(* CoDeSys 2.3.9.41 project: GermesLib_1_51.pro *)
(* Libraries: PID_Regulators.lib 6.11.19 15:29:27, Util.lib 18.5.10 15:14:28, STANDARD.LIB 4.10.05 11:14:46, IECSFC.LIB 13.4.06 15:51:28, ANALYZATION.LIB 5.10.99 09:05:06 *)

(* PLC configuration (modules and I/O channels)
Fast discrete inputs [I_SIMPLE_INPUT] node 0, in %IB0 out %QB0 {Filtrationtime = 10}
  DD1_DI0 AT %IX0.0 [BitInput] резерв
  DD1_DI1 AT %IX0.1 [BitInput] резерв
  DD1_DI2 AT %IX0.2 [BitInput] резерв
  DD1_DI3 AT %IX0.3 [BitInput] резерв
Discrete inputs [ID130] node 1, in %IB1 out %QB1 {Filtrationtime_GeneralINP = 10; Visibility = No; PinCount = 12}
  AT %IB1.0 [ByteInput] 8 discrete inputs
  AT %IB1.1 [ByteInput] 4 discrete inputs
Discrete outputs [ID131] node 2, in %IB2 out %QB2 {SafeValueByte = 0; SafeValueByteM = 0; Visibility = No; PinCount = 12}
  AT %QB2.0 [ByteOutput] 8 discrete outputs
  AT %QB2.1 [ByteOutput] 4 discrete outputs
Fast analog inputs [ID125] node 3, in %IB3 out %QB3 {Flt_Comm = 50Hz 2Por}
  DD1_AI0 AT %IR3.0 [FloatInputP] AI #1 - датчик температуры в помещении (метран) {AIN_TYPE = 4-20 mA; Peak_Filtr = 200; Flt_Ch = Off; TauRC = 10; MinFV = 0; MaxFV = 100}
  DD1_AI1 AT %IR3.1 [FloatInputP] AI #2 - расходомер FT01.01 (на входе, до отстойника) {AIN_TYPE = 4-20 mA; Peak_Filtr = 200; Flt_Ch = Off; TauRC = 10; MinFV = 0; MaxFV = 600}
  DD1_AI2 AT %IR3.2 [FloatInputP] AI #3 - расходомер FT01.02 (на выходе, после отстойника) {AIN_TYPE = 4-20 mA; Peak_Filtr = 200; Flt_Ch = Off; TauRC = 10; MinFV = 0; MaxFV = 600}
  DD1_AI3 AT %IR3.3 [FloatInputP] AI #4 - рН-метр QE01.01 (на входе, до отстойника) {AIN_TYPE = 4-20 mA; Peak_Filtr = 200; Flt_Ch = Off; TauRC = 10; MinFV = 0; MaxFV = 14}
  DD1_AI4 AT %IR3.4 [FloatInputP] AI #5 - рН-метр QE01.02 (на выходе, после отстойника) {AIN_TYPE = 4-20 mA; Peak_Filtr = 200; Flt_Ch = Off; TauRC = 10; MinFV = 0; MaxFV = 14}
  DD1_AI5 AT %IR3.5 [FloatInputP] AI #6 - сигнал от ФПК, давление на входе {AIN_TYPE = 4-20 mA; Peak_Filtr = 200; Flt_Ch = Off; TauRC = 10; MinFV = 0; MaxFV = 16}
  DD1_AI6 AT %IR3.6 [FloatInputP] AI #7 - резерв {AIN_TYPE = 4-20 mA; Peak_Filtr = 200; Flt_Ch = Off; TauRC = 10; MinFV = 0; MaxFV = 20000.0}
  DD1_AI7 AT %IR3.7 [FloatInputP] AI#8 - резерв {AIN_TYPE = 4-20 mA; Peak_Filtr = 200; Flt_Ch = Off; TauRC = 10; MinFV = 0; MaxFV = 20000.0}
  AT %IW3.8 [WordInput] AI read time (10ms)
Analog outputs [ID126] node 4, in %IB4 out %QB4
  DD1_AO0 AT %QR4.0 [FloatOutputP] AO #1 - управление ЧРП Н01.05 (поддержание расхода по расходомеру FT01.02) {AOUT_TYPE = 4-20 mA; SafeValueREAL = 0.0}
  DD1_AO1 AT %QR4.1 [FloatOutputP] AO #2 - управление ЧРП НД08.03/01 (подача флокулянта на входе, до отстойника, по FT01.01) {AOUT_TYPE = 4-20 mA; SafeValueREAL = 0.0}
  DD1_AO2 AT %QR4.2 [FloatOutputP] AO #3 - управление ЧРП НД08.03/02 (подача флокулянта на входе, до отстойника, по FT01.01) {AOUT_TYPE = 4-20 mA; SafeValueREAL = 0.0}
  DD1_AO3 AT %QR4.3 [FloatOutputP] AO #4 - управление НД05.02/01 (подача 10%NaCl из УПГ на входе, до отстойника, по FT01.01) {AOUT_TYPE = 4-20 mA; SafeValueREAL = 0.0}
Special input [ID103] node 5, in %IB5 out %QB5 {Filtrationtime = 1000; PinCount = 1; WatchDogPeriod = 400; PollPeriod = 3000; Visibility = No}
  AT %IX5.0 [BitInput] Special input
Special output [ID104] node 6, in %IB6 out %QB6 {Visibility = No; PinCount = 1}
  AT %QX6.0 [BitOutput] Special output
lastAddress AT %QD7.0 [DWordOutput] Last address
lastError AT %QW7.1 [WordOutput] Last error
RS-485-1 [COM1_USART] node 0, in %IB7.0 out %QB7.0 {CommunicationSpeed = 9600; Parity = EVEN; BitLength = 8 bits; StopLength = One stop bit; InterfaceType = RS485; FrameOriented = RTU; Timeout = 0; Visibility = No}
Universal Modbus device [ID2000] node 1, in %IB7.1 out %QB7.1 {ModuleIP = 10:0:0:102; ServiceTimeout = 20; TCPport = 502; NetMode = Serial; ModuleSlaveAddress = 2; RequestType = Both; PeriodOfService = 100; Visibility = No; RepeatCounter = 0; ByteSequence = Trace_mode}
  AT %QB7.1.0 [ComChannel] Command (0xff - Start)
DD2_DO AT %QD7.1.0.0 [DWordOutput] регистр 0, команда 0х0f
Universal Modbus device [ID2000] node 2, in %IB7.2 out %QB7.2 {ModuleIP = 10:0:0:103; ServiceTimeout = 20; TCPport = 502; NetMode = Serial; ModuleSlaveAddress = 3; RequestType = Both; PeriodOfService = 100; Visibility = No; RepeatCounter = 0; ByteSequence = Trace_mode}
  AT %QB7.2.0 [ComChannel] Command (0xff - Start)
DD3_DO AT %QD7.2.0.0 [DWordOutput]
Universal Modbus device [ID2000] node 3, in %IB7.3 out %QB7.3 {ModuleIP = 10:0:0:104; ServiceTimeout = 20; TCPport = 502; NetMode = Serial; ModuleSlaveAddress = 4; RequestType = Both; PeriodOfService = 100; Visibility = No; RepeatCounter = 0; ByteSequence = Trace_mode}
  AT %QB7.3.0 [ComChannel] Command (0xff - Start)
  32bit output module [ID2006] node 0, in %IB7.3.0 out %QB7.3.0 {ModbusAddress = 0; Command_write_regs = Force multiple coils (0x0f); Visibility = No}
    DD4_DO AT %QD7.3.0.0 [DWordOutput]
Universal Modbus device [ID2000] node 4, in %IB7.4 out %QB7.4 {ModuleIP = 10:0:0:105; ServiceTimeout = 20; TCPport = 502; NetMode = Serial; ModuleSlaveAddress = 5; RequestType = Both; PeriodOfService = 100; Visibility = No; RepeatCounter = 0; ByteSequence = Trace_mode}
  AT %QB7.4.0 [ComChannel] Command (0xff - Start)
DD5_DI AT %ID7.4.0.0 [DWordInput]
Universal Modbus device [ID2000] node 5, in %IB7.5 out %QB7.5 {ModuleIP = 10:0:0:106; ServiceTimeout = 20; TCPport = 502; NetMode = Serial; ModuleSlaveAddress = 6; RequestType = Both; PeriodOfService = 100; Visibility = No; RepeatCounter = 0; ByteSequence = Trace_mode}
  AT %QB7.5.0 [ComChannel] Command (0xff - Start)
DD6_DI AT %ID7.5.0.0 [DWordInput]
Universal Modbus device [ID2000] node 6, in %IB7.6 out %QB7.6 {ModuleIP = 10:0:0:107; ServiceTimeout = 20; TCPport = 502; NetMode = Serial; ModuleSlaveAddress = 7; RequestType = Both; PeriodOfService = 100; Visibility = No; RepeatCounter = 0; ByteSequence = Trace_mode}
  AT %QB7.6.0 [ComChannel] Command (0xff - Start)
DD7_DI AT %ID7.6.0.0 [DWordInput]
Universal Modbus device [ID2000] node 7, in %IB7.7 out %QB7.7 {ModuleIP = 10:0:0:108; ServiceTimeout = 20; TCPport = 502; NetMode = Serial; ModuleSlaveAddress = 8; RequestType = Both; PeriodOfService = 100; Visibility = No; RepeatCounter = 0; ByteSequence = Trace_mode}
  AT %QB7.7.0 [ComChannel] Command (0xff - Start)
DD8_DI AT %ID7.7.0.0 [DWordInput]
Universal Modbus device [ID2000] node 8, in %IB7.8 out %QB7.8 {ModuleIP = 10:0:0:109; ServiceTimeout = 20; TCPport = 502; NetMode = Serial; ModuleSlaveAddress = 9; RequestType = Both; PeriodOfService = 100; Visibility = No; RepeatCounter = 0; ByteSequence = Trace_mode}
  AT %QB7.8.0 [ComChannel] Command (0xff - Start)
DD9_DI AT %ID7.8.0.0 [DWordInput]
Universal Modbus device [ID2000] node 9, in %IB7.9 out %QB7.9 {ModuleIP = 10:0:0:110; ServiceTimeout = 20; TCPport = 502; NetMode = Serial; ModuleSlaveAddress = 10; RequestType = Both; PeriodOfService = 100; Visibility = No; RepeatCounter = 0; ByteSequence = Trace_mode}
  AT %QB7.9.0 [ComChannel] Command (0xff - Start)
DD10_AO0 AT %QW7.9.0.0 [WordOutput] управление 4...20мА НД05.02/02
DD10_AO1 AT %QW7.9.1.0 [WordOutput] управление 4...20мА НД06.02/01
DD10_AO2 AT %QW7.9.2.0 [WordOutput] управление 4...20мА НД06.02/02
DD10_AO3 AT %QW7.9.3.0 [WordOutput] управление 4...20мА НД06.03/01
DD10_AO4 AT %QW7.9.4.0 [WordOutput] управление 4...20мА НД06.03/02
DD10_AO5 AT %QW7.9.5.0 [WordOutput] управление 4...20мА НД07.03/01
DD10_AO6 AT %QW7.9.6.0 [WordOutput] управление 4...20мА НД07.03/02
DD10_AO7 AT %QW7.9.7.0 [WordOutput] управление 4...20мА НД08.04
Universal Modbus device [ID2000] node 10, in %IB7.10 out %QB7.10 {ModuleIP = 10:0:0:223; ServiceTimeout = 20; TCPport = 502; NetMode = Serial; ModuleSlaveAddress = 11; RequestType = By value change; PeriodOfService = 100; Visibility = No; RepeatCounter = 0; ByteSequence = Trace_mode}
  AT %QB7.10.0 [ComChannel] Command (0xff - Start)
AT %QB7.10.0.0 [ByteOutput]
Universal Modbus device [ID2000] node 11, in %IB7.11 out %QB7.11 {ModuleIP = 10:0:0:223; ServiceTimeout = 20; TCPport = 502; NetMode = Serial; ModuleSlaveAddress = 11; RequestType = By poll time; PeriodOfService = 100; Visibility = No; RepeatCounter = 0; ByteSequence = Trace_mode}
  AT %QB7.11.0 [ComChannel] Command (0xff - Start)
AT %IB7.11.0.0 [ByteInput]
Universal Modbus device [ID2000] node 12, in %IB7.12 out %QB7.12 {ModuleIP = 10:0:0:223; ServiceTimeout = 20; TCPport = 502; NetMode = Serial; ModuleSlaveAddress = 12; RequestType = By value change; PeriodOfService = 100; Visibility = No; RepeatCounter = 0; ByteSequence = Trace_mode}
  AT %QB7.12.0 [ComChannel] Command (0xff - Start)
AT %QB7.12.0.0 [ByteOutput]
Universal Modbus device [ID2000] node 13, in %IB7.13 out %QB7.13 {ModuleIP = 10:0:0:223; ServiceTimeout = 20; TCPport = 502; NetMode = Serial; ModuleSlaveAddress = 12; RequestType = By poll time; PeriodOfService = 100; Visibility = No; RepeatCounter = 0; ByteSequence = Trace_mode}
  AT %QB7.13.0 [ComChannel] Command (0xff - Start)
AT %IB7.13.0.0 [ByteInput]
AT %QD8.0 [DWordOutput] Last address
AT %QW8.1 [WordOutput] Last error
RS-232 [COM2_USART] node 0, in %IB8.0 out %QB8.0 {CommunicationSpeed = 57600; Parity = NO PARITY CHECK; BitLength = 8 bits; StopLength = One stop bit; InterfaceType = RS232; FrameOriented = RTU; Timeout = 0; Visibility = No}
AT %QB8.1.0 [ComChannel] Command (0xff - Start)
Real output module [ID2008] node 0, in %IB8.1.0 out %QB8.1.0 {ModbusAddress = 256; Command_write_regs = Preset multiple Registers (0x10); Visibility = No}
  panFT0101value AT %QD8.1.0.0 [FloatOutput]
Real output module [ID2008] node 1, in %IB8.1.1 out %QB8.1.1 {ModbusAddress = 258; Command_write_regs = Preset multiple Registers (0x10); Visibility = No}
  panQE0101value AT %QD8.1.1.0 [FloatOutput]
Real output module [ID2008] node 2, in %IB8.1.2 out %QB8.1.2 {ModbusAddress = 260; Command_write_regs = Preset multiple Registers (0x10); Visibility = No}
  panFT0102value AT %QD8.1.2.0 [FloatOutput]
Real output module [ID2008] node 3, in %IB8.1.3 out %QB8.1.3 {ModbusAddress = 262; Command_write_regs = Preset multiple Registers (0x10); Visibility = No}
  panQE0102value AT %QD8.1.3.0 [FloatOutput]
Real output module [ID2008] node 4, in %IB8.1.4 out %QB8.1.4 {ModbusAddress = 264; Command_write_regs = Preset multiple Registers (0x10); Visibility = No}
  panFPKpressureValue AT %QD8.1.4.0 [FloatOutput]
Real output module [ID2008] node 5, in %IB8.1.5 out %QB8.1.5 {ModbusAddress = 266; Command_write_regs = Preset multiple Registers (0x10); Visibility = No}
  panFQS0301total AT %QD8.1.5.0 [FloatOutput]
Real output module [ID2008] node 6, in %IB8.1.6 out %QB8.1.6 {ModbusAddress = 268; Command_write_regs = Preset multiple Registers (0x10); Visibility = No}
  panTemperature AT %QD8.1.6.0 [FloatOutput]
Register output module [ID2004] node 7, in %IB8.1.7 out %QB8.1.7 {ModbusAddress = 270; Command_write_one_reg = Write multiple registers(0x10); Visibility = No}
  panND050201workDays AT %QW8.1.7.0 [WordOutput]
Register output module [ID2004] node 8, in %IB8.1.8 out %QB8.1.8 {ModbusAddress = 271; Command_write_one_reg = Write multiple registers(0x10); Visibility = No}
  panND050201workHours AT %QW8.1.8.0 [WordOutput]
Register output module [ID2004] node 9, in %IB8.1.9 out %QB8.1.9 {ModbusAddress = 272; Command_write_one_reg = Write multiple registers(0x10); Visibility = No}
  panND050201workMinutes AT %QW8.1.9.0 [WordOutput]
Register output module [ID2004] node 10, in %IB8.1.10 out %QB8.1.10 {ModbusAddress = 273; Command_write_one_reg = Write multiple registers(0x10); Visibility = No}
  panND050201workSeconds AT %QW8.1.10.0 [WordOutput]
Register output module [ID2004] node 11, in %IB8.1.11 out %QB8.1.11 {ModbusAddress = 274; Command_write_one_reg = Write multiple registers(0x10); Visibility = No}
  panND050202workDays AT %QW8.1.11.0 [WordOutput]
Register output module [ID2004] node 12, in %IB8.1.12 out %QB8.1.12 {ModbusAddress = 275; Command_write_one_reg = Write multiple registers(0x10); Visibility = No}
  panND050202workHours AT %QW8.1.12.0 [WordOutput]
Register output module [ID2004] node 13, in %IB8.1.13 out %QB8.1.13 {ModbusAddress = 276; Command_write_one_reg = Write multiple registers(0x10); Visibility = No}
  panND050202workMinutes AT %QW8.1.13.0 [WordOutput]
Register output module [ID2004] node 14, in %IB8.1.14 out %QB8.1.14 {ModbusAddress = 277; Command_write_one_reg = Write multiple registers(0x10); Visibility = No}
  panND050202workSeconds AT %QW8.1.14.0 [WordOutput]
Register output module [ID2004] node 15, in %IB8.1.15 out %QB8.1.15 {ModbusAddress = 278; Command_write_one_reg = Write multiple registers(0x10); Visibility = No}
  panND0502counterP1 AT %QW8.1.15.0 [WordOutput]
Register output module [ID2004] node 16, in %IB8.1.16 out %QB8.1.16 {ModbusAddress = 279; Command_write_one_reg = Write multiple registers(0x10); Visibility = No}
  panND0502counterP2 AT %QW8.1.16.0 [WordOutput]
Register output module [ID2004] node 17, in %IB8.1.17 out %QB8.1.17 {ModbusAddress = 280; Command_write_one_reg = Write multiple registers(0x10); Visibility = No}
  panND060201workDays AT %QW8.1.17.0 [WordOutput]
Register output module [ID2004] node 18, in %IB8.1.18 out %QB8.1.18 {ModbusAddress = 281; Command_write_one_reg = Write multiple registers(0x10); Visibility = No}
  panND060201workHours AT %QW8.1.18.0 [WordOutput]
Register output module [ID2004] node 19, in %IB8.1.19 out %QB8.1.19 {ModbusAddress = 282; Command_write_one_reg = Write multiple registers(0x10); Visibility = No}
  panND060201workMinutes AT %QW8.1.19.0 [WordOutput]
Register output module [ID2004] node 20, in %IB8.1.20 out %QB8.1.20 {ModbusAddress = 283; Command_write_one_reg = Write multiple registers(0x10); Visibility = No}
  panND060201workSeconds AT %QW8.1.20.0 [WordOutput]
Register output module [ID2004] node 21, in %IB8.1.21 out %QB8.1.21 {ModbusAddress = 284; Command_write_one_reg = Write multiple registers(0x10); Visibility = No}
  panND060202workDays AT %QW8.1.21.0 [WordOutput]
Register output module [ID2004] node 22, in %IB8.1.22 out %QB8.1.22 {ModbusAddress = 285; Command_write_one_reg = Write multiple registers(0x10); Visibility = No}
  panND060202workHours AT %QW8.1.22.0 [WordOutput]
Register output module [ID2004] node 23, in %IB8.1.23 out %QB8.1.23 {ModbusAddress = 286; Command_write_one_reg = Write multiple registers(0x10); Visibility = No}
  panND060202workMinutes AT %QW8.1.23.0 [WordOutput]
Register output module [ID2004] node 24, in %IB8.1.24 out %QB8.1.24 {ModbusAddress = 287; Command_write_one_reg = Write multiple registers(0x10); Visibility = No}
  panND060202workSeconds AT %QW8.1.24.0 [WordOutput]
Register output module [ID2004] node 25, in %IB8.1.25 out %QB8.1.25 {ModbusAddress = 288; Command_write_one_reg = Write multiple registers(0x10); Visibility = No}
  panND0602counterP1 AT %QW8.1.25.0 [WordOutput]
Register output module [ID2004] node 26, in %IB8.1.26 out %QB8.1.26 {ModbusAddress = 289; Command_write_one_reg = Write multiple registers(0x10); Visibility = No}
  panND0602counterP2 AT %QW8.1.26.0 [WordOutput]
Register output module [ID2004] node 27, in %IB8.1.27 out %QB8.1.27 {ModbusAddress = 290; Command_write_one_reg = Write multiple registers(0x10); Visibility = No}
  panND060301workDays AT %QW8.1.27.0 [WordOutput]
Register output module [ID2004] node 28, in %IB8.1.28 out %QB8.1.28 {ModbusAddress = 291; Command_write_one_reg = Write multiple registers(0x10); Visibility = No}
  panND060301workHours AT %QW8.1.28.0 [WordOutput]
Register output module [ID2004] node 29, in %IB8.1.29 out %QB8.1.29 {ModbusAddress = 292; Command_write_one_reg = Write multiple registers(0x10); Visibility = No}
  panND060301workMinutes AT %QW8.1.29.0 [WordOutput]
Register output module [ID2004] node 30, in %IB8.1.30 out %QB8.1.30 {ModbusAddress = 293; Command_write_one_reg = Write multiple registers(0x10); Visibility = No}
  panND060301workSeconds AT %QW8.1.30.0 [WordOutput]
Register output module [ID2004] node 31, in %IB8.1.31 out %QB8.1.31 {ModbusAddress = 294; Command_write_one_reg = Write multiple registers(0x10); Visibility = No}
  panND060302workDays AT %QW8.1.31.0 [WordOutput]
Register output module [ID2004] node 32, in %IB8.1.32 out %QB8.1.32 {ModbusAddress = 295; Command_write_one_reg = Write multiple registers(0x10); Visibility = No}
  panND060302workHours AT %QW8.1.32.0 [WordOutput]
Register output module [ID2004] node 33, in %IB8.1.33 out %QB8.1.33 {ModbusAddress = 296; Command_write_one_reg = Write multiple registers(0x10); Visibility = No}
  panND060302workMinutes AT %QW8.1.33.0 [WordOutput]
Register output module [ID2004] node 34, in %IB8.1.34 out %QB8.1.34 {ModbusAddress = 297; Command_write_one_reg = Write multiple registers(0x10); Visibility = No}
  panND060302workSeconds AT %QW8.1.34.0 [WordOutput]
Register output module [ID2004] node 35, in %IB8.1.35 out %QB8.1.35 {ModbusAddress = 298; Command_write_one_reg = Write multiple registers(0x10); Visibility = No}
  panND0603counterP1 AT %QW8.1.35.0 [WordOutput]
Register output module [ID2004] node 36, in %IB8.1.36 out %QB8.1.36 {ModbusAddress = 299; Command_write_one_reg = Write multiple registers(0x10); Visibility = No}
  panND0603counterP2 AT %QW8.1.36.0 [WordOutput]
Register output module [ID2004] node 37, in %IB8.1.37 out %QB8.1.37 {ModbusAddress = 300; Command_write_one_reg = Write multiple registers(0x10); Visibility = No}
  panND070301workDays AT %QW8.1.37.0 [WordOutput]
Register output module [ID2004] node 38, in %IB8.1.38 out %QB8.1.38 {ModbusAddress = 301; Command_write_one_reg = Write multiple registers(0x10); Visibility = No}
  panND070301workHours AT %QW8.1.38.0 [WordOutput]
Register output module [ID2004] node 39, in %IB8.1.39 out %QB8.1.39 {ModbusAddress = 302; Command_write_one_reg = Write multiple registers(0x10); Visibility = No}
  panND070301workMinutes AT %QW8.1.39.0 [WordOutput]
Register output module [ID2004] node 40, in %IB8.1.40 out %QB8.1.40 {ModbusAddress = 303; Command_write_one_reg = Write multiple registers(0x10); Visibility = No}
  panND070301workSeconds AT %QW8.1.40.0 [WordOutput]
Register output module [ID2004] node 41, in %IB8.1.41 out %QB8.1.41 {ModbusAddress = 304; Command_write_one_reg = Write multiple registers(0x10); Visibility = No}
  panND070302workDays AT %QW8.1.41.0 [WordOutput]
Register output module [ID2004] node 42, in %IB8.1.42 out %QB8.1.42 {ModbusAddress = 305; Command_write_one_reg = Write multiple registers(0x10); Visibility = No}
  panND070302workHours AT %QW8.1.42.0 [WordOutput]
Register output module [ID2004] node 43, in %IB8.1.43 out %QB8.1.43 {ModbusAddress = 306; Command_write_one_reg = Write multiple registers(0x10); Visibility = No}
  panND070302workMinutes AT %QW8.1.43.0 [WordOutput]
Register output module [ID2004] node 44, in %IB8.1.44 out %QB8.1.44 {ModbusAddress = 307; Command_write_one_reg = Write multiple registers(0x10); Visibility = No}
  panND070302workSeconds AT %QW8.1.44.0 [WordOutput]
Register output module [ID2004] node 45, in %IB8.1.45 out %QB8.1.45 {ModbusAddress = 308; Command_write_one_reg = Write multiple registers(0x10); Visibility = No}
  panND0703counterP1 AT %QW8.1.45.0 [WordOutput]
Register output module [ID2004] node 46, in %IB8.1.46 out %QB8.1.46 {ModbusAddress = 309; Command_write_one_reg = Write multiple registers(0x10); Visibility = No}
  panND0703counterP2 AT %QW8.1.46.0 [WordOutput]
Register output module [ID2004] node 47, in %IB8.1.47 out %QB8.1.47 {ModbusAddress = 310; Command_write_one_reg = Write multiple registers(0x10); Visibility = No}
  panND080301workDays AT %QW8.1.47.0 [WordOutput]
Register output module [ID2004] node 48, in %IB8.1.48 out %QB8.1.48 {ModbusAddress = 311; Command_write_one_reg = Write multiple registers(0x10); Visibility = No}
  panND080301workHours AT %QW8.1.48.0 [WordOutput]
Register output module [ID2004] node 49, in %IB8.1.49 out %QB8.1.49 {ModbusAddress = 312; Command_write_one_reg = Write multiple registers(0x10); Visibility = No}
  panND080301workMinutes AT %QW8.1.49.0 [WordOutput]
Register output module [ID2004] node 50, in %IB8.1.50 out %QB8.1.50 {ModbusAddress = 313; Command_write_one_reg = Write multiple registers(0x10); Visibility = No}
  panND080301workSeconds AT %QW8.1.50.0 [WordOutput]
Register output module [ID2004] node 51, in %IB8.1.51 out %QB8.1.51 {ModbusAddress = 314; Command_write_one_reg = Write multiple registers(0x10); Visibility = No}
  panND080302workDays AT %QW8.1.51.0 [WordOutput]
Register output module [ID2004] node 52, in %IB8.1.52 out %QB8.1.52 {ModbusAddress = 315; Command_write_one_reg = Write multiple registers(0x10); Visibility = No}
  panND080302workHours AT %QW8.1.52.0 [WordOutput]
Register output module [ID2004] node 53, in %IB8.1.53 out %QB8.1.53 {ModbusAddress = 316; Command_write_one_reg = Write multiple registers(0x10); Visibility = No}
  panND080302workMinutes AT %QW8.1.53.0 [WordOutput]
Register output module [ID2004] node 54, in %IB8.1.54 out %QB8.1.54 {ModbusAddress = 317; Command_write_one_reg = Write multiple registers(0x10); Visibility = No}
  panND080302workSeconds AT %QW8.1.54.0 [WordOutput]
Register output module [ID2004] node 55, in %IB8.1.55 out %QB8.1.55 {ModbusAddress = 318; Command_write_one_reg = Write multiple registers(0x10); Visibility = No}
  panND0803counterP1 AT %QW8.1.55.0 [WordOutput]
Register output module [ID2004] node 56, in %IB8.1.56 out %QB8.1.56 {ModbusAddress = 319; Command_write_one_reg = Write multiple registers(0x10); Visibility = No}
  panND0803counterP2 AT %QW8.1.56.0 [WordOutput]
Register output module [ID2004] node 57, in %IB8.1.57 out %QB8.1.57 {ModbusAddress = 320; Command_write_one_reg = Write multiple registers(0x10); Visibility = No}
  panN010501workDays AT %QW8.1.57.0 [WordOutput]
Register output module [ID2004] node 58, in %IB8.1.58 out %QB8.1.58 {ModbusAddress = 321; Command_write_one_reg = Write multiple registers(0x10); Visibility = No}
  panN010501workHours AT %QW8.1.58.0 [WordOutput]
Register output module [ID2004] node 59, in %IB8.1.59 out %QB8.1.59 {ModbusAddress = 322; Command_write_one_reg = Write multiple registers(0x10); Visibility = No}
  panN010501workMinutes AT %QW8.1.59.0 [WordOutput]
Register output module [ID2004] node 60, in %IB8.1.60 out %QB8.1.60 {ModbusAddress = 323; Command_write_one_reg = Write multiple registers(0x10); Visibility = No}
  panN010501workSeconds AT %QW8.1.60.0 [WordOutput]
Register output module [ID2004] node 61, in %IB8.1.61 out %QB8.1.61 {ModbusAddress = 324; Command_write_one_reg = Write multiple registers(0x10); Visibility = No}
  panN010502workDays AT %QW8.1.61.0 [WordOutput]
Register output module [ID2004] node 62, in %IB8.1.62 out %QB8.1.62 {ModbusAddress = 325; Command_write_one_reg = Write multiple registers(0x10); Visibility = No}
  panN010502workHours AT %QW8.1.62.0 [WordOutput]
Register output module [ID2004] node 63, in %IB8.1.63 out %QB8.1.63 {ModbusAddress = 326; Command_write_one_reg = Write multiple registers(0x10); Visibility = No}
  panN010502workMinutes AT %QW8.1.63.0 [WordOutput]
Register output module [ID2004] node 64, in %IB8.1.64 out %QB8.1.64 {ModbusAddress = 327; Command_write_one_reg = Write multiple registers(0x10); Visibility = No}
  panN010502workSeconds AT %QW8.1.64.0 [WordOutput]
Register output module [ID2004] node 65, in %IB8.1.65 out %QB8.1.65 {ModbusAddress = 328; Command_write_one_reg = Write multiple registers(0x10); Visibility = No}
  panN0105counterP1 AT %QW8.1.65.0 [WordOutput]
Register output module [ID2004] node 66, in %IB8.1.66 out %QB8.1.66 {ModbusAddress = 329; Command_write_one_reg = Write multiple registers(0x10); Visibility = No}
  panN0105counterP2 AT %QW8.1.66.0 [WordOutput]
Register output module [ID2004] node 67, in %IB8.1.67 out %QB8.1.67 {ModbusAddress = 330; Command_write_one_reg = Write multiple registers(0x10); Visibility = No}
  panN020401workDays AT %QW8.1.67.0 [WordOutput]
Register output module [ID2004] node 68, in %IB8.1.68 out %QB8.1.68 {ModbusAddress = 331; Command_write_one_reg = Write multiple registers(0x10); Visibility = No}
  panN020401workHours AT %QW8.1.68.0 [WordOutput]
Register output module [ID2004] node 69, in %IB8.1.69 out %QB8.1.69 {ModbusAddress = 332; Command_write_one_reg = Write multiple registers(0x10); Visibility = No}
  panN020401workMinutes AT %QW8.1.69.0 [WordOutput]
Register output module [ID2004] node 70, in %IB8.1.70 out %QB8.1.70 {ModbusAddress = 333; Command_write_one_reg = Write multiple registers(0x10); Visibility = No}
  panN020401workSeconds AT %QW8.1.70.0 [WordOutput]
Register output module [ID2004] node 71, in %IB8.1.71 out %QB8.1.71 {ModbusAddress = 334; Command_write_one_reg = Write multiple registers(0x10); Visibility = No}
  panN020402workDays AT %QW8.1.71.0 [WordOutput]
Register output module [ID2004] node 72, in %IB8.1.72 out %QB8.1.72 {ModbusAddress = 335; Command_write_one_reg = Write multiple registers(0x10); Visibility = No}
  panN020402workHours AT %QW8.1.72.0 [WordOutput]
Register output module [ID2004] node 73, in %IB8.1.73 out %QB8.1.73 {ModbusAddress = 336; Command_write_one_reg = Write multiple registers(0x10); Visibility = No}
  panN020402workMinutes AT %QW8.1.73.0 [WordOutput]
Register output module [ID2004] node 74, in %IB8.1.74 out %QB8.1.74 {ModbusAddress = 337; Command_write_one_reg = Write multiple registers(0x10); Visibility = No}
  panN020402workSeconds AT %QW8.1.74.0 [WordOutput]
Register output module [ID2004] node 75, in %IB8.1.75 out %QB8.1.75 {ModbusAddress = 338; Command_write_one_reg = Write multiple registers(0x10); Visibility = No}
  panN0204counterP1 AT %QW8.1.75.0 [WordOutput]
Register output module [ID2004] node 76, in %IB8.1.76 out %QB8.1.76 {ModbusAddress = 339; Command_write_one_reg = Write multiple registers(0x10); Visibility = No}
  panN0204counterP2 AT %QW8.1.76.0 [WordOutput]
Register output module [ID2004] node 77, in %IB8.1.77 out %QB8.1.77 {ModbusAddress = 340; Command_write_one_reg = Write multiple registers(0x10); Visibility = No}
  panN040401workDays AT %QW8.1.77.0 [WordOutput]
Register output module [ID2004] node 78, in %IB8.1.78 out %QB8.1.78 {ModbusAddress = 341; Command_write_one_reg = Write multiple registers(0x10); Visibility = No}
  panN040401workHours AT %QW8.1.78.0 [WordOutput]
Register output module [ID2004] node 79, in %IB8.1.79 out %QB8.1.79 {ModbusAddress = 342; Command_write_one_reg = Write multiple registers(0x10); Visibility = No}
  panN040401workMinutes AT %QW8.1.79.0 [WordOutput]
Register output module [ID2004] node 80, in %IB8.1.80 out %QB8.1.80 {ModbusAddress = 343; Command_write_one_reg = Write multiple registers(0x10); Visibility = No}
  panN040401workSeconds AT %QW8.1.80.0 [WordOutput]
Register output module [ID2004] node 81, in %IB8.1.81 out %QB8.1.81 {ModbusAddress = 344; Command_write_one_reg = Write multiple registers(0x10); Visibility = No}
  panN040402workDays AT %QW8.1.81.0 [WordOutput]
Register output module [ID2004] node 82, in %IB8.1.82 out %QB8.1.82 {ModbusAddress = 345; Command_write_one_reg = Write multiple registers(0x10); Visibility = No}
  panN040402workHours AT %QW8.1.82.0 [WordOutput]
Register output module [ID2004] node 83, in %IB8.1.83 out %QB8.1.83 {ModbusAddress = 346; Command_write_one_reg = Write multiple registers(0x10); Visibility = No}
  panN040402workMinutes AT %QW8.1.83.0 [WordOutput]
Register output module [ID2004] node 84, in %IB8.1.84 out %QB8.1.84 {ModbusAddress = 347; Command_write_one_reg = Write multiple registers(0x10); Visibility = No}
  panN040402workSeconds AT %QW8.1.84.0 [WordOutput]
Register output module [ID2004] node 85, in %IB8.1.85 out %QB8.1.85 {ModbusAddress = 348; Command_write_one_reg = Write multiple registers(0x10); Visibility = No}
  panN0404counterP1 AT %QW8.1.85.0 [WordOutput]
Register output module [ID2004] node 86, in %IB8.1.86 out %QB8.1.86 {ModbusAddress = 349; Command_write_one_reg = Write multiple registers(0x10); Visibility = No}
  panN0404counterP2 AT %QW8.1.86.0 [WordOutput]
Register output module [ID2004] node 87, in %IB8.1.87 out %QB8.1.87 {ModbusAddress = 350; Command_write_one_reg = Write multiple registers(0x10); Visibility = No}
  panUFO030101workDays AT %QW8.1.87.0 [WordOutput]
Register output module [ID2004] node 88, in %IB8.1.88 out %QB8.1.88 {ModbusAddress = 351; Command_write_one_reg = Write multiple registers(0x10); Visibility = No}
  panUFO030101workHours AT %QW8.1.88.0 [WordOutput]
Register output module [ID2004] node 89, in %IB8.1.89 out %QB8.1.89 {ModbusAddress = 352; Command_write_one_reg = Write multiple registers(0x10); Visibility = No}
  panUFO030101workMinutes AT %QW8.1.89.0 [WordOutput]
Register output module [ID2004] node 90, in %IB8.1.90 out %QB8.1.90 {ModbusAddress = 353; Command_write_one_reg = Write multiple registers(0x10); Visibility = No}
  panUFO030101workSeconds AT %QW8.1.90.0 [WordOutput]
Register output module [ID2004] node 91, in %IB8.1.91 out %QB8.1.91 {ModbusAddress = 354; Command_write_one_reg = Write multiple registers(0x10); Visibility = No}
  panUFO030102workDays AT %QW8.1.91.0 [WordOutput]
Register output module [ID2004] node 92, in %IB8.1.92 out %QB8.1.92 {ModbusAddress = 355; Command_write_one_reg = Write multiple registers(0x10); Visibility = No}
  panUFO030102workHours AT %QW8.1.92.0 [WordOutput]
Register output module [ID2004] node 93, in %IB8.1.93 out %QB8.1.93 {ModbusAddress = 356; Command_write_one_reg = Write multiple registers(0x10); Visibility = No}
  panUFO030102workMinutes AT %QW8.1.93.0 [WordOutput]
Register output module [ID2004] node 94, in %IB8.1.94 out %QB8.1.94 {ModbusAddress = 357; Command_write_one_reg = Write multiple registers(0x10); Visibility = No}
  panUFO030102workSeconds AT %QW8.1.94.0 [WordOutput]
Register output module [ID2004] node 95, in %IB8.1.95 out %QB8.1.95 {ModbusAddress = 358; Command_write_one_reg = Write multiple registers(0x10); Visibility = No}
  panUFO0301counterP1 AT %QW8.1.95.0 [WordOutput]
Register output module [ID2004] node 96, in %IB8.1.96 out %QB8.1.96 {ModbusAddress = 359; Command_write_one_reg = Write multiple registers(0x10); Visibility = No}
  panUFO0301counterP2 AT %QW8.1.96.0 [WordOutput]
panVolumeToRegen AT %QD8.1.97.0 [FloatOutput]
8 bit output module [ID2002] node 98, in %IB8.1.98 out %QB8.1.98 {ModbusAddress = 256; Command_write_byte = Force multiply coils (0x0f); Visibility = No}
  AT %QB8.1.98.0 [ByteOutput]
8 bit output module [ID2002] node 99, in %IB8.1.99 out %QB8.1.99 {ModbusAddress = 264; Command_write_byte = Force multiply coils (0x0f); Visibility = No}
  AT %QB8.1.99.0 [ByteOutput]
8 bit output module [ID2002] node 100, in %IB8.1.100 out %QB8.1.100 {ModbusAddress = 272; Command_write_byte = Force multiply coils (0x0f); Visibility = No}
  AT %QB8.1.100.0 [ByteOutput]
8 bit output module [ID2002] node 101, in %IB8.1.101 out %QB8.1.101 {ModbusAddress = 280; Command_write_byte = Force multiply coils (0x0f); Visibility = No}
  AT %QB8.1.101.0 [ByteOutput]
8 bit output module [ID2002] node 102, in %IB8.1.102 out %QB8.1.102 {ModbusAddress = 288; Command_write_byte = Force multiply coils (0x0f); Visibility = No}
  AT %QB8.1.102.0 [ByteOutput]
8 bit output module [ID2002] node 103, in %IB8.1.103 out %QB8.1.103 {ModbusAddress = 296; Command_write_byte = Force multiply coils (0x0f); Visibility = No}
  AT %QB8.1.103.0 [ByteOutput]
8 bit output module [ID2002] node 104, in %IB8.1.104 out %QB8.1.104 {ModbusAddress = 304; Command_write_byte = Force multiply coils (0x0f); Visibility = No}
  AT %QB8.1.104.0 [ByteOutput]
8 bit output module [ID2002] node 105, in %IB8.1.105 out %QB8.1.105 {ModbusAddress = 312; Command_write_byte = Force multiply coils (0x0f); Visibility = No}
  AT %QB8.1.105.0 [ByteOutput]
8 bit output module [ID2002] node 106, in %IB8.1.106 out %QB8.1.106 {ModbusAddress = 320; Command_write_byte = Force multiply coils (0x0f); Visibility = No}
  AT %QB8.1.106.0 [ByteOutput]
8 bit output module [ID2002] node 107, in %IB8.1.107 out %QB8.1.107 {ModbusAddress = 328; Command_write_byte = Force multiply coils (0x0f); Visibility = No}
  AT %QB8.1.107.0 [ByteOutput]
8 bit output module [ID2002] node 108, in %IB8.1.108 out %QB8.1.108 {ModbusAddress = 336; Command_write_byte = Force multiply coils (0x0f); Visibility = No}
  AT %QB8.1.108.0 [ByteOutput]
8 bit output module [ID2002] node 109, in %IB8.1.109 out %QB8.1.109 {ModbusAddress = 344; Command_write_byte = Force multiply coils (0x0f); Visibility = No}
  AT %QB8.1.109.0 [ByteOutput]
8 bit output module [ID2002] node 110, in %IB8.1.110 out %QB8.1.110 {ModbusAddress = 352; Command_write_byte = Force multiply coils (0x0f); Visibility = No}
  AT %QB8.1.110.0 [ByteOutput]
8 bit output module [ID2002] node 111, in %IB8.1.111 out %QB8.1.111 {ModbusAddress = 360; Command_write_byte = Force multiply coils (0x0f); Visibility = No}
  AT %QB8.1.111.0 [ByteOutput]
8 bit output module [ID2002] node 112, in %IB8.1.112 out %QB8.1.112 {ModbusAddress = 368; Command_write_byte = Force multiply coils (0x0f); Visibility = No}
  AT %QB8.1.112.0 [ByteOutput]
8 bit output module [ID2002] node 113, in %IB8.1.113 out %QB8.1.113 {ModbusAddress = 376; Command_write_byte = Force multiply coils (0x0f); Visibility = No}
  AT %QB8.1.113.0 [ByteOutput]
8 bit output module [ID2002] node 114, in %IB8.1.114 out %QB8.1.114 {ModbusAddress = 384; Command_write_byte = Force multiply coils (0x0f); Visibility = No}
  AT %QB8.1.114.0 [ByteOutput]
8 bit output module [ID2002] node 115, in %IB8.1.115 out %QB8.1.115 {ModbusAddress = 392; Command_write_byte = Force multiply coils (0x0f); Visibility = No}
  AT %QB8.1.115.0 [ByteOutput]
8 bit output module [ID2002] node 116, in %IB8.1.116 out %QB8.1.116 {ModbusAddress = 400; Command_write_byte = Force multiply coils (0x0f); Visibility = No}
  AT %QB8.1.116.0 [ByteOutput]
8 bit output module [ID2002] node 117, in %IB8.1.117 out %QB8.1.117 {ModbusAddress = 408; Command_write_byte = Force multiply coils (0x0f); Visibility = No}
  AT %QB8.1.117.0 [ByteOutput]
8 bit output module [ID2002] node 118, in %IB8.1.118 out %QB8.1.118 {ModbusAddress = 416; Command_write_byte = Force multiply coils (0x0f); Visibility = No}
  AT %QB8.1.118.0 [ByteOutput]
8 bit output module [ID2002] node 119, in %IB8.1.119 out %QB8.1.119 {ModbusAddress = 424; Command_write_byte = Force multiply coils (0x0f); Visibility = No}
  AT %QB8.1.119.0 [ByteOutput]
8 bit output module [ID2002] node 120, in %IB8.1.120 out %QB8.1.120 {ModbusAddress = 432; Command_write_byte = Force multiply coils (0x0f); Visibility = No}
  AT %QB8.1.120.0 [ByteOutput]
8 bit output module [ID2002] node 121, in %IB8.1.121 out %QB8.1.121 {ModbusAddress = 440; Command_write_byte = Force multiply coils (0x0f); Visibility = No}
  AT %QB8.1.121.0 [ByteOutput]
8 bit output module [ID2002] node 122, in %IB8.1.122 out %QB8.1.122 {ModbusAddress = 448; Command_write_byte = Force multiply coils (0x0f); Visibility = No}
  AT %QB8.1.122.0 [ByteOutput]
8 bit output module [ID2002] node 123, in %IB8.1.123 out %QB8.1.123 {ModbusAddress = 456; Command_write_byte = Force multiply coils (0x0f); Visibility = No}
  AT %QB8.1.123.0 [ByteOutput]
8 bit output module [ID2002] node 124, in %IB8.1.124 out %QB8.1.124 {ModbusAddress = 464; Command_write_byte = Force multiply coils (0x0f); Visibility = No}
  AT %QB8.1.124.0 [ByteOutput]
8 bit output module [ID2002] node 125, in %IB8.1.125 out %QB8.1.125 {ModbusAddress = 472; Command_write_byte = Force multiply coils (0x0f); Visibility = No}
  AT %QB8.1.125.0 [ByteOutput]
8 bit output module [ID2002] node 126, in %IB8.1.126 out %QB8.1.126 {ModbusAddress = 480; Command_write_byte = Force multiply coils (0x0f); Visibility = No}
  AT %QB8.1.126.0 [ByteOutput]
8 bit output module [ID2002] node 127, in %IB8.1.127 out %QB8.1.127 {ModbusAddress = 488; Command_write_byte = Force multiply coils (0x0f); Visibility = No}
  AT %QB8.1.127.0 [ByteOutput]
8 bit output module [ID2002] node 128, in %IB8.1.128 out %QB8.1.128 {ModbusAddress = 496; Command_write_byte = Force multiply coils (0x0f); Visibility = No}
  AT %QB8.1.128.0 [ByteOutput]
8 bit output module [ID2002] node 129, in %IB8.1.129 out %QB8.1.129 {ModbusAddress = 504; Command_write_byte = Force multiply coils (0x0f); Visibility = No}
  AT %QB8.1.129.0 [ByteOutput]
8 bit output module [ID2002] node 130, in %IB8.1.130 out %QB8.1.130 {ModbusAddress = 512; Command_write_byte = Force multiply coils (0x0f); Visibility = No}
  AT %QB8.1.130.0 [ByteOutput]
8 bit output module [ID2002] node 131, in %IB8.1.131 out %QB8.1.131 {ModbusAddress = 520; Command_write_byte = Force multiply coils (0x0f); Visibility = No}
  AT %QB8.1.131.0 [ByteOutput]
8 bit output module [ID2002] node 132, in %IB8.1.132 out %QB8.1.132 {ModbusAddress = 528; Command_write_byte = Force multiply coils (0x0f); Visibility = No}
  AT %QB8.1.132.0 [ByteOutput]
8 bit output module [ID2002] node 133, in %IB8.1.133 out %QB8.1.133 {ModbusAddress = 632; Command_write_byte = Force multiply coils (0x0f); Visibility = No}
  AT %QB8.1.133.0 [ByteOutput]
  AT %QB8.1.134.0 [ByteOutput]
Universal Modbus device [ID2000] node 2, in %IB8.2 out %QB8.2 {ModuleIP = 10:0:0:223; ServiceTimeout = 150; TCPport = 502; NetMode = Serial; ModuleSlaveAddress = 1; RequestType = By poll time; PeriodOfService = 10; Visibility = No; RepeatCounter = 0; ByteSequence = Native}
  AT %QB8.2.0 [ComChannel] Command (0xff - Start)
  8 bit input module [ID2001] node 0, in %IB8.2.0 out %QB8.2.0 {ModbusAddress = 536; Command_read_byte = Read coils status (0x01); Visibility = No}
    AT %IB8.2.0.0 [ByteInput]
  8 bit input module [ID2001] node 1, in %IB8.2.1 out %QB8.2.1 {ModbusAddress = 544; Command_read_byte = Read coils status (0x01); Visibility = No}
    AT %IB8.2.1.0 [ByteInput]
  8 bit input module [ID2001] node 2, in %IB8.2.2 out %QB8.2.2 {ModbusAddress = 552; Command_read_byte = Read coils status (0x01); Visibility = No}
    AT %IB8.2.2.0 [ByteInput]
  8 bit input module [ID2001] node 3, in %IB8.2.3 out %QB8.2.3 {ModbusAddress = 560; Command_read_byte = Read coils status (0x01); Visibility = No}
    AT %IB8.2.3.0 [ByteInput]
  8 bit input module [ID2001] node 4, in %IB8.2.4 out %QB8.2.4 {ModbusAddress = 568; Command_read_byte = Read coils status (0x01); Visibility = No}
    AT %IB8.2.4.0 [ByteInput]
  8 bit input module [ID2001] node 5, in %IB8.2.5 out %QB8.2.5 {ModbusAddress = 576; Command_read_byte = Read coils status (0x01); Visibility = No}
    AT %IB8.2.5.0 [ByteInput]
  8 bit input module [ID2001] node 6, in %IB8.2.6 out %QB8.2.6 {ModbusAddress = 584; Command_read_byte = Read coils status (0x01); Visibility = No}
    AT %IB8.2.6.0 [ByteInput]
  8 bit input module [ID2001] node 7, in %IB8.2.7 out %QB8.2.7 {ModbusAddress = 592; Command_read_byte = Read coils status (0x01); Visibility = No}
    AT %IB8.2.7.0 [ByteInput]
  8 bit input module [ID2001] node 8, in %IB8.2.8 out %QB8.2.8 {ModbusAddress = 600; Command_read_byte = Read coils status (0x01); Visibility = No}
    AT %IB8.2.8.0 [ByteInput]
  8 bit input module [ID2001] node 9, in %IB8.2.9 out %QB8.2.9 {ModbusAddress = 608; Command_read_byte = Read coils status (0x01); Visibility = No}
    AT %IB8.2.9.0 [ByteInput]
  8 bit input module [ID2001] node 10, in %IB8.2.10 out %QB8.2.10 {ModbusAddress = 616; Command_read_byte = Read coils status (0x01); Visibility = No}
    AT %IB8.2.10.0 [ByteInput]
  8 bit input module [ID2001] node 11, in %IB8.2.11 out %QB8.2.11 {ModbusAddress = 624; Command_read_byte = Read coils status (0x01); Visibility = No}
    AT %IB8.2.11.0 [ByteInput]
  Real input module [ID2007] node 12, in %IB8.2.12 out %QB8.2.12 {ModbusAddress = 10256; Command_read_regs = Read holding Registers  (0x03); Visibility = No}
    panTimeToOpenCloseValve AT %ID8.2.12.0 [FloatInput]
  Register input module [ID2003] node 13, in %IB8.2.13 out %QB8.2.13 {ModbusAddress = 10258; Command_read_regs = Read holding Registers  (0x03); Visibility = No}
    panMaxTemperature AT %IW8.2.13.0 [WordInput]
  Register input module [ID2003] node 14, in %IB8.2.14 out %QB8.2.14 {ModbusAddress = 10259; Command_read_regs = Read holding Registers  (0x03); Visibility = No}
    panMinTemperature AT %IW8.2.14.0 [WordInput]
  Real input module [ID2007] node 15, in %IB8.2.15 out %QB8.2.15 {ModbusAddress = 10260; Command_read_regs = Read holding Registers  (0x03); Visibility = No}
    panND0502setMaxDosVal AT %ID8.2.15.0 [FloatInput]
  Real input module [ID2007] node 16, in %IB8.2.16 out %QB8.2.16 {ModbusAddress = 10262; Command_read_regs = Read holding Registers  (0x03); Visibility = No}
    panND0502setKoefProp AT %ID8.2.16.0 [FloatInput]
  Real input module [ID2007] node 17, in %IB8.2.17 out %QB8.2.17 {ModbusAddress = 10264; Command_read_regs = Read holding Registers  (0x03); Visibility = No}
    panND0602setMaxDosVal AT %ID8.2.17.0 [FloatInput]
  Real input module [ID2007] node 18, in %IB8.2.18 out %QB8.2.18 {ModbusAddress = 10266; Command_read_regs = Read holding Registers  (0x03); Visibility = No}
    panND0602setKoefProp AT %ID8.2.18.0 [FloatInput]
  Real input module [ID2007] node 19, in %IB8.2.19 out %QB8.2.19 {ModbusAddress = 10268; Command_read_regs = Read holding Registers  (0x03); Visibility = No}
    panND0603setMaxDosVal AT %ID8.2.19.0 [FloatInput]
  Real input module [ID2007] node 20, in %IB8.2.20 out %QB8.2.20 {ModbusAddress = 10270; Command_read_regs = Read holding Registers  (0x03); Visibility = No}
    panND0603setKoefProp AT %ID8.2.20.0 [FloatInput]
  Real input module [ID2007] node 21, in %IB8.2.21 out %QB8.2.21 {ModbusAddress = 10272; Command_read_regs = Read holding Registers  (0x03); Visibility = No}
    panND0703pHsetValue AT %ID8.2.21.0 [FloatInput]
  Real input module [ID2007] node 22, in %IB8.2.22 out %QB8.2.22 {ModbusAddress = 10274; Command_read_regs = Read holding Registers  (0x03); Visibility = No}
    panND0703YoutManual AT %ID8.2.22.0 [FloatInput]
  Real input module [ID2007] node 23, in %IB8.2.23 out %QB8.2.23 {ModbusAddress = 10276; Command_read_regs = Read holding Registers  (0x03); Visibility = No}
    panND0703koeffI AT %ID8.2.23.0 [FloatInput]
  Real input module [ID2007] node 24, in %IB8.2.24 out %QB8.2.24 {ModbusAddress = 10278; Command_read_regs = Read holding Registers  (0x03); Visibility = No}
    panND0703koeffD AT %ID8.2.24.0 [FloatInput]
  Real input module [ID2007] node 25, in %IB8.2.25 out %QB8.2.25 {ModbusAddress = 10280; Command_read_regs = Read holding Registers  (0x03); Visibility = No}
    panND0703koeffP AT %ID8.2.25.0 [FloatInput]
  Real input module [ID2007] node 26, in %IB8.2.26 out %QB8.2.26 {ModbusAddress = 10282; Command_read_regs = Read holding Registers  (0x03); Visibility = No}
    panND0803setMaxDosVal AT %ID8.2.26.0 [FloatInput]
  Real input module [ID2007] node 27, in %IB8.2.27 out %QB8.2.27 {ModbusAddress = 10284; Command_read_regs = Read holding Registers  (0x03); Visibility = No}
    panND0803setKoefProp AT %ID8.2.27.0 [FloatInput]
  Register input module [ID2003] node 28, in %IB8.2.28 out %QB8.2.28 {ModbusAddress = 10286; Command_read_regs = Read holding Registers  (0x03); Visibility = No}
    panND0804doseValue AT %IW8.2.28.0 [WordInput]
  Real input module [ID2007] node 29, in %IB8.2.29 out %QB8.2.29 {ModbusAddress = 10287; Command_read_regs = Read holding Registers  (0x03); Visibility = No}
    panN0105flowSetValue AT %ID8.2.29.0 [FloatInput]
  Real input module [ID2007] node 30, in %IB8.2.30 out %QB8.2.30 {ModbusAddress = 10289; Command_read_regs = Read holding Registers  (0x03); Visibility = No}
    panN0105YoutManual AT %ID8.2.30.0 [FloatInput]
  Real input module [ID2007] node 31, in %IB8.2.31 out %QB8.2.31 {ModbusAddress = 10291; Command_read_regs = Read holding Registers  (0x03); Visibility = No}
    panN0105koeffI AT %ID8.2.31.0 [FloatInput]
  Real input module [ID2007] node 32, in %IB8.2.32 out %QB8.2.32 {ModbusAddress = 10293; Command_read_regs = Read holding Registers  (0x03); Visibility = No}
    panN0105koeffD AT %ID8.2.32.0 [FloatInput]
  Real input module [ID2007] node 33, in %IB8.2.33 out %QB8.2.33 {ModbusAddress = 10295; Command_read_regs = Read holding Registers  (0x03); Visibility = No}
    panN0105koeffP AT %ID8.2.33.0 [FloatInput]
  Real input module [ID2007] node 34, in %IB8.2.34 out %QB8.2.34 {ModbusAddress = 10297; Command_read_regs = Read holding Registers  (0x03); Visibility = No}
    panFQS0301impulsValue AT %ID8.2.34.0 [FloatInput]
  Real input module [ID2007] node 35, in %IB8.2.35 out %QB8.2.35 {ModbusAddress = 10299; Command_read_regs = Read holding Registers  (0x03); Visibility = No}
    panFQS0301correction AT %ID8.2.35.0 [FloatInput]
  Real input module [ID2007] node 36, in %IB8.2.36 out %QB8.2.36 {ModbusAddress = 10301; Command_read_regs = Read holding Registers  (0x03); Visibility = No}
    panFPKtimeToWork AT %ID8.2.36.0 [FloatInput]
  Real input module [ID2007] node 37, in %IB8.2.37 out %QB8.2.37 {ModbusAddress = 10303; Command_read_regs = Read holding Registers  (0x03); Visibility = No}
    panFPKnotStartedTime AT %ID8.2.37.0 [FloatInput]
  Real input module [ID2007] node 38, in %IB8.2.38 out %QB8.2.38 {ModbusAddress = 10305; Command_read_regs = Read holding Registers  (0x03); Visibility = No}
    panFPKmaxPressureValue AT %ID8.2.38.0 [FloatInput]
  Real input module [ID2007] node 39, in %IB8.2.39 out %QB8.2.39 {ModbusAddress = 10307; Command_read_regs = Read holding Registers  (0x03); Visibility = No}
    panFilterValueToRegen AT %ID8.2.39.0 [FloatInput]
ModBus (slave) [MODBUS_ID400] node 9, in %IB9 out %QB9 {SlaveIdentificator = 1; Visibility = No}
  Modbus [MODBUS_ID302] node 0, in %IB9.0 out %QB9.0
    TCP [TCP_ID221] node 0, in %IB9.0.0 out %QB9.0.0 {RemotePort = 502; Visibility = No}
  Float [Float] node 1, in %IB9.1 out %QB9.1
    remFT0101value AT %QD9.1.0 [FloatOutput] Расходомер на входе
  Float [Float] node 2, in %IB9.2 out %QB9.2
    remFQS0301totalAmount AT %QD9.2.0 [FloatOutput] Счетчик очищенных стоков
  Float [Float] node 3, in %IB9.3 out %QB9.3
    remTemperatureValue AT %QD9.3.0 [FloatOutput] Температура в помещении
  8 bits [8Bit] node 4, in %IB9.4 out %QB9.4
    AT %QB9.4.0 [ByteOutput]
  8 bits [8Bit] node 5, in %IB9.5 out %QB9.5
    AT %QB9.5.0 [ByteOutput]
*)

(* POU PLC_PRG, CFC *)
PROGRAM PLC_PRG
VAR
	test: RichThreePumpManager;
	start1: BOOL;
	start2: BOOL;
	p1main: BOOL;
	p2main: BOOL;
	p3main: BOOL;
	bycounter: BOOL;
	byworktime: BOOL;
	alarm1in: BOOL;
	alarm2in: BOOL;
	alarm3in: BOOL;
	alarmreset: BOOL;
	start1man: BOOL;
	start2man: BOOL;
	start3man: BOOL;
	resetwt1: BOOL;
	resetwt2: BOOL;
	resetwt3: BOOL;
	resetcount1: BOOL;
	resetcount2: BOOL;
	resetcount3: BOOL;
	delayrepeatedstart: UINT;
	delaystart2: UINT;
	statp1main: BOOL;
	statp2main: BOOL;
	statp3main: BOOL;
	statbycount: BOOL;
	statbywt: BOOL;
	started1: BOOL;
	started2: BOOL;
	started3: BOOL;
	counter1: UDINT;
	counter2: UDINT;
	counter3: UDINT;
	days1: UINT;
	hours1: UINT;
	minutes1: UINT;
	seconds1: UINT;
	days2: UINT;
	hours2: UINT;
	minutes2: UINT;
	seconds2: UINT;
	days3: UINT;
	hours3: UINT;
	minutes3: UINT;
	seconds3: UINT;
	nxtStartP1: UINT;
	nxtStartP2: UINT;
	nxtStartP3: UINT;
	alarm1out: BOOL;
	alarm2out: BOOL;
	alarm3out: BOOL;
END_VAR
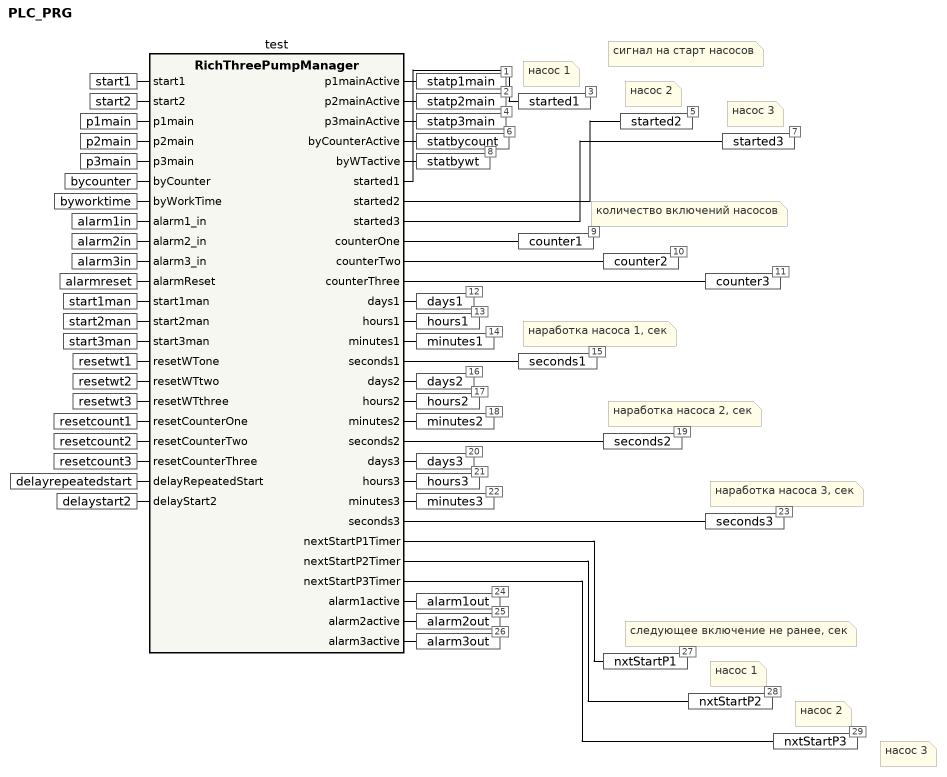
_CFC_ (* Continuous Function Chart, elements in execution order *)
(* сигнал на старт насосов *)
(* количество включений насосов *)
(* наработка насоса 1, сек *)
(* следующее включение не ранее, сек *)
(* насос 1 *)
(* насос 3 *)
(* наработка насоса 2, сек *)
(* наработка насоса 3, сек *)
(* насос 2 *)
(* насос 1 *)
(* насос 3 *)
(* насос 2 *)
#0 test:RichThreePumpManager(start1: start1, start2: start2, p1main: p1main, p2main: p2main, p3main: p3main, byCounter: bycounter, byWorkTime: byworktime, alarm1_in: alarm1in, alarm2_in: alarm2in, alarm3_in: alarm3in, alarmReset: alarmreset, start1man: start1man, start2man: start2man, start3man: start3man, resetWTone: resetwt1, resetWTtwo: resetwt2, resetWTthree: resetwt3, resetCounterOne: resetcount1, resetCounterTwo: resetcount2, resetCounterThree: resetcount3, delayRepeatedStart: delayrepeatedstart, delayStart2: delaystart2)
#1 statp1main <= #0.p1mainActive
#2 statp2main <= #0.p2mainActive
#3 started1 <= #0.started1
#4 statp3main <= #0.p3mainActive
#5 started2 <= #0.started2
#6 statbycount <= #0.byCounterActive
#7 started3 <= #0.started3
#8 statbywt <= #0.byWTactive
#9 counter1 <= #0.counterOne
#10 counter2 <= #0.counterTwo
#11 counter3 <= #0.counterThree
#12 days1 <= #0.days1
#13 hours1 <= #0.hours1
#14 minutes1 <= #0.minutes1
#15 seconds1 <= #0.seconds1
#16 days2 <= #0.days2
#17 hours2 <= #0.hours2
#18 minutes2 <= #0.minutes2
#19 seconds2 <= #0.seconds2
#20 days3 <= #0.days3
#21 hours3 <= #0.hours3
#22 minutes3 <= #0.minutes3
#23 seconds3 <= #0.seconds3
#24 alarm1out <= #0.alarm1active
#25 alarm2out <= #0.alarm2active
#26 alarm3out <= #0.alarm3active
#27 nxtStartP1 <= #0.nextStartP1Timer
#28 nxtStartP2 <= #0.nextStartP2Timer
#29 nxtStartP3 <= #0.nextStartP3Timer
_END_CFC_
(* the same logic as Structured Text *)
(* сигнал на старт насосов *)
(* количество включений насосов *)
(* наработка насоса 1, сек *)
(* следующее включение не ранее, сек *)
(* насос 1 *)
(* насос 3 *)
(* наработка насоса 2, сек *)
(* наработка насоса 3, сек *)
(* насос 2 *)
(* насос 1 *)
(* насос 3 *)
(* насос 2 *)
test(start1 := start1, start2 := start2, p1main := p1main, p2main := p2main, p3main := p3main, byCounter := bycounter, byWorkTime := byworktime, alarm1_in := alarm1in, alarm2_in := alarm2in, alarm3_in := alarm3in, alarmReset := alarmreset, start1man := start1man, start2man := start2man, start3man := start3man, resetWTone := resetwt1, resetWTtwo := resetwt2, resetWTthree := resetwt3, resetCounterOne := resetcount1, resetCounterTwo := resetcount2, resetCounterThree := resetcount3, delayRepeatedStart := delayrepeatedstart, delayStart2 := delaystart2);
statp1main := test.p1mainActive;
statp2main := test.p2mainActive;
started1 := test.started1;
statp3main := test.p3mainActive;
started2 := test.started2;
statbycount := test.byCounterActive;
started3 := test.started3;
statbywt := test.byWTactive;
counter1 := test.counterOne;
counter2 := test.counterTwo;
counter3 := test.counterThree;
days1 := test.days1;
hours1 := test.hours1;
minutes1 := test.minutes1;
seconds1 := test.seconds1;
days2 := test.days2;
hours2 := test.hours2;
minutes2 := test.minutes2;
seconds2 := test.seconds2;
days3 := test.days3;
hours3 := test.hours3;
minutes3 := test.minutes3;
seconds3 := test.seconds3;
alarm1out := test.alarm1active;
alarm2out := test.alarm2active;
alarm3out := test.alarm3active;
nxtStartP1 := test.nextStartP1Timer;
nxtStartP2 := test.nextStartP2Timer;
nxtStartP3 := test.nextStartP3Timer;
END_PROGRAM

(* POU RichThreePumpManager, CFC *)
FUNCTION_BLOCK RichThreePumpManager
VAR_INPUT
	start1: BOOL;
	start2: BOOL;
	p1main: BOOL;
	p2main: BOOL;
	p3main: BOOL;
	byCounter: BOOL;
	byWorkTime: BOOL;
	alarm1_in: BOOL;
	alarm2_in: BOOL;
	alarm3_in: BOOL;
	alarmReset: BOOL;
	start1man: BOOL;
	start2man: BOOL;
	start3man: BOOL;
	resetWTone: BOOL;
	resetWTtwo: BOOL;
	resetWTthree: BOOL;
	resetCounterOne: BOOL;
	resetCounterTwo: BOOL;
	resetCounterThree: BOOL;
	delayRepeatedStart: UINT;		(*задержка повторного пуска, сек.*)
	delayStart2: UINT;		(*задержка пуска второго после пуска первого, сек*)
END_VAR
VAR_OUTPUT
	p1mainActive: BOOL;
	p2mainActive: BOOL;
	p3mainActive: BOOL;
	byCounterActive: BOOL;
	byWTactive: BOOL;
	started1: BOOL;
	started2: BOOL;
	started3: BOOL;
	counterOne: UDINT;
	counterTwo: UDINT;
	counterThree: UDINT;
	days1: UINT;
	hours1: UINT;
	minutes1: UINT;
	seconds1: UINT;
	days2: UINT;
	hours2: UINT;
	minutes2: UINT;
	seconds2: UINT;
	days3: UINT;
	hours3: UINT;
	minutes3: UINT;
	seconds3: UINT;
	nextStartP1Timer: UINT;
	nextStartP2Timer: UINT;
	nextStartP3Timer: UINT;
	alarm1active: BOOL;
	alarm2active: BOOL;
	alarm3active: BOOL;
END_VAR
VAR
	ctpr: ChooseThreePumpRegime;
	slft: StartLessFromThree;
	alarmTrig1: RS;
	alarmTrig2: RS;
	alarmTrig3: RS;
	stp: SimpleThreePump;
	frsp1: FastRepeatedStartProtection;
	frsp2: FastRepeatedStartProtection;
	frsp3: FastRepeatedStartProtection;
	pps1: PulsePerSec;
	pps2: PulsePerSec;
	pps3: PulsePerSec;
	icwt1: ImpulsCounter;
	icw2: ImpulsCounter;
	icwt3: ImpulsCounter;
	ts1: TimeSeparator;
	ts2: TimeSeparator;
	ts3: TimeSeparator;
	ic1: ImpulsCounter;
	ic2: ImpulsCounter;
	ic3: ImpulsCounter;
	WorkTimeOne: UDINT;
	WorkTimeTwo: UDINT;
	WorkTimeThree: UDINT;
END_VAR
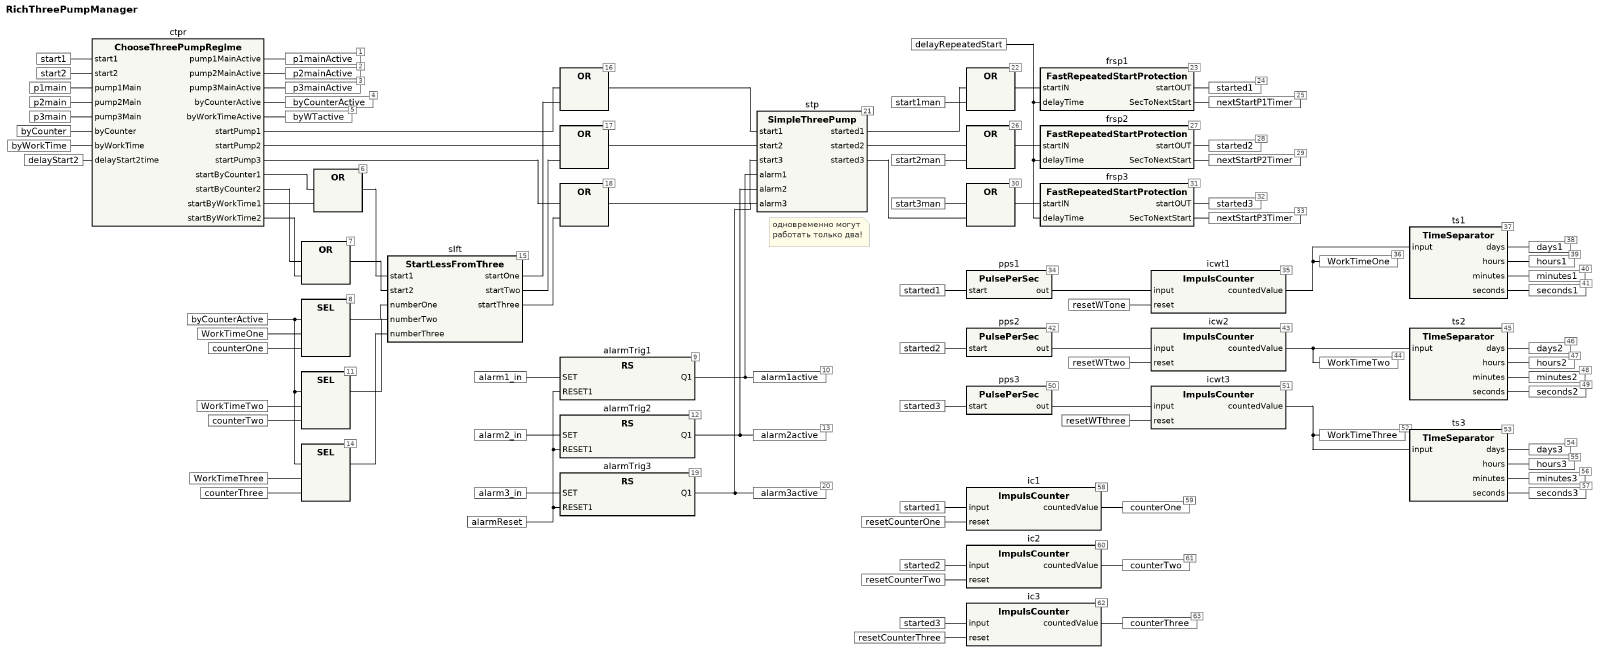
_CFC_ (* Continuous Function Chart, elements in execution order *)
(* одновременно могут / работать только два! *)
#0 ctpr:ChooseThreePumpRegime(start1: start1, start2: start2, pump1Main: p1main, pump2Main: p2main, pump3Main: p3main, byCounter: byCounter, byWorkTime: byWorkTime, delayStart2time: delayStart2)
#1 p1mainActive <= #0.pump1MainActive
#2 p2mainActive <= #0.pump2MainActive
#3 p3mainActive <= #0.pump3MainActive
#4 byCounterActive <= #0.byCounterActive
#5 byWTactive <= #0.byWorkTimeActive
#6 OR(#0.startByCounter1, #0.startByWorkTime1)
#7 OR(#0.startByCounter2, #0.startByWorkTime2)
#8 SEL(byCounterActive, WorkTimeOne, counterOne)
#9 alarmTrig1:RS(SET: alarm1_in, RESET1: alarmReset)
#10 alarm1active <= #9.Q1
#11 SEL(byCounterActive, WorkTimeTwo, counterTwo)
#12 alarmTrig2:RS(SET: alarm2_in, RESET1: alarmReset)
#13 alarm2active <= #12.Q1
#14 SEL(byCounterActive, WorkTimeThree, counterThree)
#15 slft:StartLessFromThree(start1: #6, start2: #7, numberOne: #8, numberTwo: #11, numberThree: #14)
#16 OR(#0.startPump1, #15.startOne)
#17 OR(#0.startPump2, #15.startTwo)
#18 OR(#0.startPump3, #15.startThree)
#19 alarmTrig3:RS(SET: alarm3_in, RESET1: alarmReset)
#20 alarm3active <= #19.Q1
#21 stp:SimpleThreePump(start1: #16, start2: #17, start3: #18, alarm1: #9.Q1, alarm2: #12.Q1, alarm3: #19.Q1)
#22 OR(#21.started1, start1man)
#23 frsp1:FastRepeatedStartProtection(startIN: #22, delayTime: delayRepeatedStart)
#24 started1 <= #23.startOUT
#25 nextStartP1Timer <= #23.SecToNextStart
#26 OR(#21.started2, start2man)
#27 frsp2:FastRepeatedStartProtection(startIN: #26, delayTime: delayRepeatedStart)
#28 started2 <= #27.startOUT
#29 nextStartP2Timer <= #27.SecToNextStart
#30 OR(start3man, #21.started3)
#31 frsp3:FastRepeatedStartProtection(startIN: #30, delayTime: delayRepeatedStart)
#32 started3 <= #31.startOUT
#33 nextStartP3Timer <= #31.SecToNextStart
#34 pps1:PulsePerSec(start: started1)
#35 icwt1:ImpulsCounter(input: #34.out, reset: resetWTone)
#36 WorkTimeOne <= #35.countedValue
#37 ts1:TimeSeparator(input: #35.countedValue)
#38 days1 <= #37.days
#39 hours1 <= #37.hours
#40 minutes1 <= #37.minutes
#41 seconds1 <= #37.seconds
#42 pps2:PulsePerSec(start: started2)
#43 icw2:ImpulsCounter(input: #42.out, reset: resetWTtwo)
#44 WorkTimeTwo <= #43.countedValue
#45 ts2:TimeSeparator(input: #43.countedValue)
#46 days2 <= #45.days
#47 hours2 <= #45.hours
#48 minutes2 <= #45.minutes
#49 seconds2 <= #45.seconds
#50 pps3:PulsePerSec(start: started3)
#51 icwt3:ImpulsCounter(input: #50.out, reset: resetWTthree)
#52 WorkTimeThree <= #51.countedValue
#53 ts3:TimeSeparator(input: #51.countedValue)
#54 days3 <= #53.days
#55 hours3 <= #53.hours
#56 minutes3 <= #53.minutes
#57 seconds3 <= #53.seconds
#58 ic1:ImpulsCounter(input: started1, reset: resetCounterOne)
#59 counterOne <= #58.countedValue
#60 ic2:ImpulsCounter(input: started2, reset: resetCounterTwo)
#61 counterTwo <= #60.countedValue
#62 ic3:ImpulsCounter(input: started3, reset: resetCounterThree)
#63 counterThree <= #62.countedValue
_END_CFC_
(* the same logic as Structured Text *)
(* одновременно могут / работать только два! *)
ctpr(start1 := start1, start2 := start2, pump1Main := p1main, pump2Main := p2main, pump3Main := p3main, byCounter := byCounter, byWorkTime := byWorkTime, delayStart2time := delayStart2);
p1mainActive := ctpr.pump1MainActive;
p2mainActive := ctpr.pump2MainActive;
p3mainActive := ctpr.pump3MainActive;
byCounterActive := ctpr.byCounterActive;
byWTactive := ctpr.byWorkTimeActive;
alarmTrig1(SET := alarm1_in, RESET1 := alarmReset);
alarm1active := alarmTrig1.Q1;
alarmTrig2(SET := alarm2_in, RESET1 := alarmReset);
alarm2active := alarmTrig2.Q1;
slft(start1 := ctpr.startByCounter1 OR ctpr.startByWorkTime1, start2 := ctpr.startByCounter2 OR ctpr.startByWorkTime2, numberOne := SEL(byCounterActive, WorkTimeOne, counterOne), numberTwo := SEL(byCounterActive, WorkTimeTwo, counterTwo), numberThree := SEL(byCounterActive, WorkTimeThree, counterThree));
alarmTrig3(SET := alarm3_in, RESET1 := alarmReset);
alarm3active := alarmTrig3.Q1;
stp(start1 := ctpr.startPump1 OR slft.startOne, start2 := ctpr.startPump2 OR slft.startTwo, start3 := ctpr.startPump3 OR slft.startThree, alarm1 := alarmTrig1.Q1, alarm2 := alarmTrig2.Q1, alarm3 := alarmTrig3.Q1);
frsp1(startIN := stp.started1 OR start1man, delayTime := delayRepeatedStart);
started1 := frsp1.startOUT;
nextStartP1Timer := frsp1.SecToNextStart;
frsp2(startIN := stp.started2 OR start2man, delayTime := delayRepeatedStart);
started2 := frsp2.startOUT;
nextStartP2Timer := frsp2.SecToNextStart;
frsp3(startIN := start3man OR stp.started3, delayTime := delayRepeatedStart);
started3 := frsp3.startOUT;
nextStartP3Timer := frsp3.SecToNextStart;
pps1(start := started1);
icwt1(input := pps1.out, reset := resetWTone);
WorkTimeOne := icwt1.countedValue;
ts1(input := icwt1.countedValue);
days1 := ts1.days;
hours1 := ts1.hours;
minutes1 := ts1.minutes;
seconds1 := ts1.seconds;
pps2(start := started2);
icw2(input := pps2.out, reset := resetWTtwo);
WorkTimeTwo := icw2.countedValue;
ts2(input := icw2.countedValue);
days2 := ts2.days;
hours2 := ts2.hours;
minutes2 := ts2.minutes;
seconds2 := ts2.seconds;
pps3(start := started3);
icwt3(input := pps3.out, reset := resetWTthree);
WorkTimeThree := icwt3.countedValue;
ts3(input := icwt3.countedValue);
days3 := ts3.days;
hours3 := ts3.hours;
minutes3 := ts3.minutes;
seconds3 := ts3.seconds;
ic1(input := started1, reset := resetCounterOne);
counterOne := ic1.countedValue;
ic2(input := started2, reset := resetCounterTwo);
counterTwo := ic2.countedValue;
ic3(input := started3, reset := resetCounterThree);
counterThree := ic3.countedValue;
END_FUNCTION_BLOCK

(* POU ChooseThreePumpRegime, CFC *)
FUNCTION_BLOCK ChooseThreePumpRegime
VAR
	pump1RStrig: RS;		(*Триггер-защелка выбора режима с главным первым насосом.*)
	pump2RStrig: RS;		(*Триггер-защелка выбора режима с главным вторым насосом.*)
	pump3RStrig: RS;		(*Триггер-защелка выбора режима с главным третьим насосом.*)
	byCounterRStrig: RS;		(*Триггер-защелка выбора режима с запуском по количеству включений.*)
	byWorkTimeRStrig: RS;		(*Триггер-защелка выбора режима с запуском по наработке.*)
	Pump1MainDetector: R_TRIG;		(*Детектор переднего фронта включения режима, когда главный насос - первый.
Для сброса остальных значений.*)
	Pump2MainDetector: R_TRIG;		(*Детектор переднего фронта включения режима, когда главный насос - второй.
Для сброса остальных значений.*)
	Pump3MainDetector: R_TRIG;		(*Детектор переднего фронта включения режима, когда главный насос - третий.
Для сброса остальных значений.*)
	ByCounterDetector: R_TRIG;		(*Детектор переднего фронта включения режима по количеству включений.
Для сброса остальных значений.*)
	ByWorkTimeDetector: R_TRIG;		(*Детектор переднего фронта включения режима по наработке.
Для сброса остальных значений.*)
	tonToStart1: TON;
	tonToStart2: TON;
	tonToStart3: TON;
	tonToStart4: TON;
	tonToStart5: TON;
END_VAR
VAR_INPUT
	start1: BOOL;		(*Сигнал на включение одного  насоса.
Активируется выход согласно выбранного режима.*)
	start2: BOOL;		(*Сигнал на включение второго насоса.
Активируется выход согласно выбранного режима.*)
	pump1Main: BOOL;		(*Режим: первый насос главный. Включать импульсом.*)
	pump2Main: BOOL;		(*Режим: второй насос главный. Включать импульсом.*)
	pump3Main: BOOL;		(*Режим: третий насос главный. Включать импульсом.*)
	byCounter: BOOL;		(*Режим: запуск по количеству включений.
Включится с меньшим количеством стартов. Включать импульсом.*)
	byWorkTime: BOOL;		(*Режим: запуск по наработке.
Включится насос с меньшей наработкой. Включать импульсом.*)
	delayStart2time: UINT;		(*время задержки пуска второго после подачи сигнала на пуск первого, сек.*)
END_VAR
VAR_OUTPUT
	pump1MainActive: BOOL;		(*Активный режим: первый насос главный.*)
	pump2MainActive: BOOL;		(*Активный режим: второй насос главный.*)
	pump3MainActive: BOOL;		(*Активный режим: третий насос главный.*)
	byCounterActive: BOOL;		(*Активный режим: включение по количеству запусков.*)
	byWorkTimeActive: BOOL;		(*Активный режим: по наработке.*)
	startPump1: BOOL;		(*Запуск первого насоса.*)
	startPump2: BOOL;		(*Запуск второго насоса.*)
	startPump3: BOOL;		(*Запуск третьего насоса.*)
	startByCounter1: BOOL;		(*Запуск насоса по количеству стартов.
			Запустится с меньшим. Если одинаково, то - первый.*)
	startByCounter2: BOOL;		(*Запуск насоса по количеству стартов.
			Запустится с меньшим. Если одинаково, то - первый.*)
	startByWorkTime1: BOOL;		(*Запуск по наработке.
			Включится с меньшей. Если одинаково, то - первый.*)
	startByWorkTime2: BOOL;		(*Запуск по наработке.
			Включится с меньшей. Если одинаково, то - первый.*)
END_VAR
VAR (* helpers for the ST form of the networks *)
	_t96 : BOOL;
	_t196 : BOOL;
	_t182 : TIME;
	_t197 : BOOL;
	_t198 : BOOL;
	_t116 : BOOL;
	_en121 : BOOL;
	_t121 : BOOL;
	_en128 : BOOL;
	_t128 : BOOL;
	_en159 : BOOL;
	_t159 : BOOL;
	_en135 : BOOL;
	_t135 : BOOL;
	_en142 : BOOL;
	_t142 : BOOL;
END_VAR
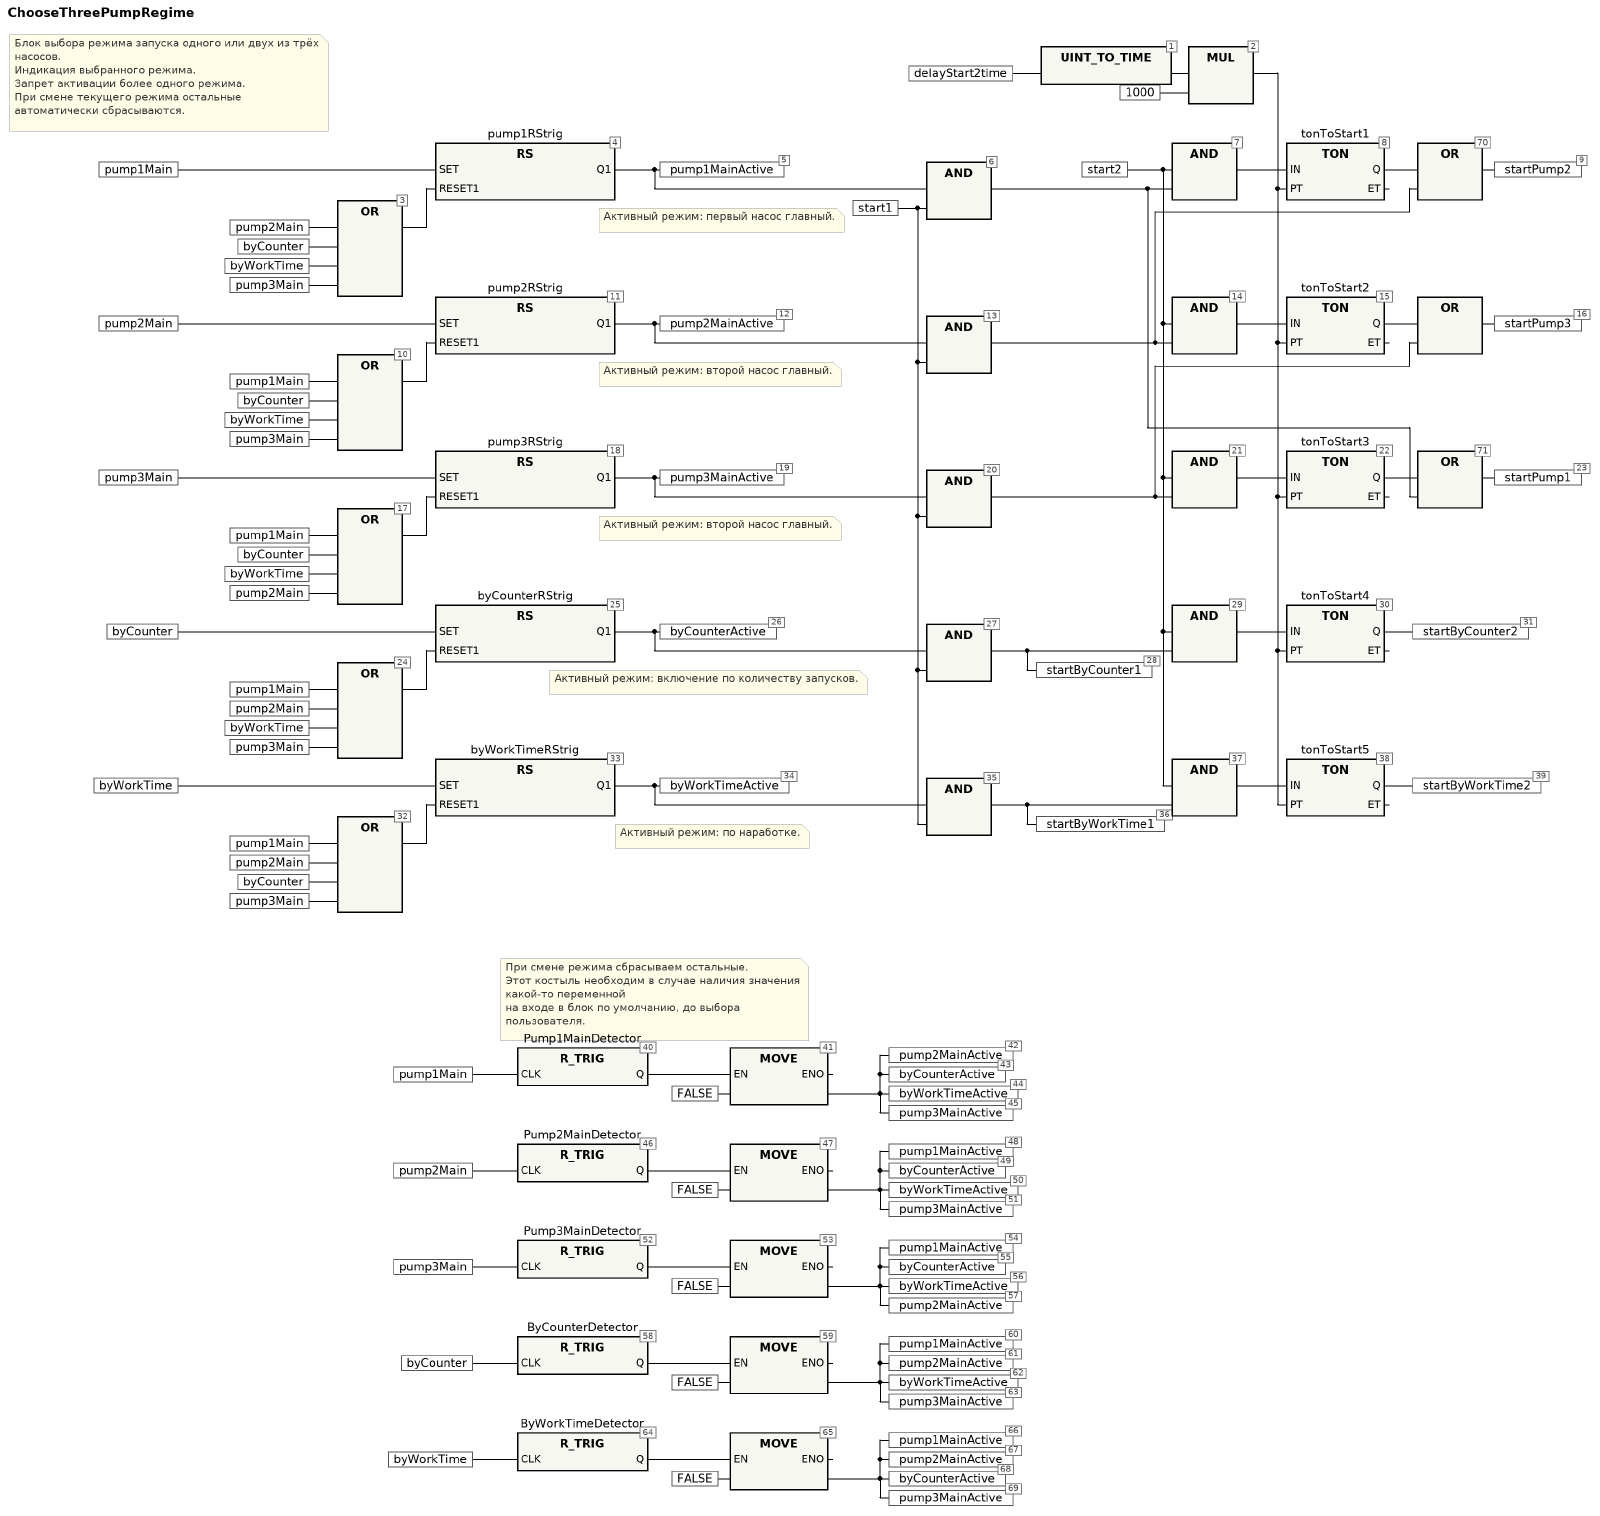
_CFC_ (* Continuous Function Chart, elements in execution order *)
(* Активный режим: второй насос главный. *)
(* Блок выбора режима запуска одного или двух из трёх насосов. / Индикация выбранного режима. / Запрет активации более одного режима. / При смене текущего режима остальные автоматически сбрасываются. *)
(* Активный режим: первый насос главный. *)
(* Активный режим: включение по количеству запусков. *)
(* Активный режим: по наработке. *)
(* Активный режим: второй насос главный. *)
(* При смене режима сбрасываем остальные. / Этот костыль необходим в случае наличия значения какой-то переменной / на входе в блок по умолчанию, до выбора пользователя. *)
#0 OR(#15.Q, #20)
#1 UINT_TO_TIME(delayStart2time)
#2 MUL(#1, 1000)
#3 OR(pump2Main, byCounter, byWorkTime, pump3Main)
#4 pump1RStrig:RS(SET: pump1Main, RESET1: #3)
#5 pump1MainActive <= #4.Q1
#6 AND(#4.Q1, start1)
#7 AND(start2, #6)
#8 tonToStart1:TON(IN: #7, PT: #2)
#9 startPump2 <= #70
#10 OR(pump1Main, byCounter, byWorkTime, pump3Main)
#11 pump2RStrig:RS(SET: pump2Main, RESET1: #10)
#12 pump2MainActive <= #11.Q1
#13 AND(#11.Q1, start1)
#14 AND(start2, #13)
#15 tonToStart2:TON(IN: #14, PT: #2)
#16 startPump3 <= #0
#17 OR(pump1Main, byCounter, byWorkTime, pump2Main)
#18 pump3RStrig:RS(SET: pump3Main, RESET1: #17)
#19 pump3MainActive <= #18.Q1
#20 AND(#18.Q1, start1)
#21 AND(start2, #20)
#22 tonToStart3:TON(IN: #21, PT: #2)
#23 startPump1 <= #71
#24 OR(pump1Main, pump2Main, byWorkTime, pump3Main)
#25 byCounterRStrig:RS(SET: byCounter, RESET1: #24)
#26 byCounterActive <= #25.Q1
#27 AND(#25.Q1, start1)
#28 startByCounter1 <= #27
#29 AND(start2, #27)
#30 tonToStart4:TON(IN: #29, PT: #2)
#31 startByCounter2 <= #30.Q
#32 OR(pump1Main, pump2Main, byCounter, pump3Main)
#33 byWorkTimeRStrig:RS(SET: byWorkTime, RESET1: #32)
#34 byWorkTimeActive <= #33.Q1
#35 AND(#33.Q1, start1)
#36 startByWorkTime1 <= #35
#37 AND(start2, #35)
#38 tonToStart5:TON(IN: #37, PT: #2)
#39 startByWorkTime2 <= #38.Q
#40 Pump1MainDetector:R_TRIG(CLK: pump1Main)
#41 MOVE(EN: #40.Q, FALSE)
#42 pump2MainActive <= #41
#43 byCounterActive <= #41
#44 byWorkTimeActive <= #41
#45 pump3MainActive <= #41
#46 Pump2MainDetector:R_TRIG(CLK: pump2Main)
#47 MOVE(EN: #46.Q, FALSE)
#48 pump1MainActive <= #47
#49 byCounterActive <= #47
#50 byWorkTimeActive <= #47
#51 pump3MainActive <= #47
#52 Pump3MainDetector:R_TRIG(CLK: pump3Main)
#53 MOVE(EN: #52.Q, FALSE)
#54 pump1MainActive <= #53
#55 byCounterActive <= #53
#56 byWorkTimeActive <= #53
#57 pump2MainActive <= #53
#58 ByCounterDetector:R_TRIG(CLK: byCounter)
#59 MOVE(EN: #58.Q, FALSE)
#60 pump1MainActive <= #59
#61 pump2MainActive <= #59
#62 byWorkTimeActive <= #59
#63 pump3MainActive <= #59
#64 ByWorkTimeDetector:R_TRIG(CLK: byWorkTime)
#65 MOVE(EN: #64.Q, FALSE)
#66 pump1MainActive <= #65
#67 pump2MainActive <= #65
#68 byCounterActive <= #65
#69 pump3MainActive <= #65
#70 OR(#8.Q, #13)
#71 OR(#22.Q, #6)
_END_CFC_
(* the same logic as Structured Text *)
(* Активный режим: второй насос главный. *)
(* Блок выбора режима запуска одного или двух из трёх насосов. / Индикация выбранного режима. / Запрет активации более одного режима. / При смене текущего режима остальные автоматически сбрасываются. *)
(* Активный режим: первый насос главный. *)
(* Активный режим: включение по количеству запусков. *)
(* Активный режим: по наработке. *)
(* Активный режим: второй насос главный. *)
(* При смене режима сбрасываем остальные. / Этот костыль необходим в случае наличия значения какой-то переменной / на входе в блок по умолчанию, до выбора пользователя. *)
_t196 := tonToStart2.Q OR _t96;
_t182 := UINT_TO_TIME(delayStart2time) * 1000;
pump1RStrig(SET := pump1Main, RESET1 := pump2Main OR byCounter OR byWorkTime OR pump3Main);
pump1MainActive := pump1RStrig.Q1;
tonToStart1(IN := start2 AND (pump1RStrig.Q1 AND start1), PT := _t182);
startPump2 := _t197;
pump2RStrig(SET := pump2Main, RESET1 := pump1Main OR byCounter OR byWorkTime OR pump3Main);
pump2MainActive := pump2RStrig.Q1;
tonToStart2(IN := start2 AND (pump2RStrig.Q1 AND start1), PT := _t182);
startPump3 := _t196;
pump3RStrig(SET := pump3Main, RESET1 := pump1Main OR byCounter OR byWorkTime OR pump2Main);
pump3MainActive := pump3RStrig.Q1;
_t96 := pump3RStrig.Q1 AND start1;
tonToStart3(IN := start2 AND _t96, PT := _t182);
startPump1 := _t198;
byCounterRStrig(SET := byCounter, RESET1 := pump1Main OR pump2Main OR byWorkTime OR pump3Main);
byCounterActive := byCounterRStrig.Q1;
startByCounter1 := byCounterRStrig.Q1 AND start1;
tonToStart4(IN := start2 AND (byCounterRStrig.Q1 AND start1), PT := _t182);
startByCounter2 := tonToStart4.Q;
byWorkTimeRStrig(SET := byWorkTime, RESET1 := pump1Main OR pump2Main OR byCounter OR pump3Main);
byWorkTimeActive := byWorkTimeRStrig.Q1;
_t116 := byWorkTimeRStrig.Q1 AND start1;
startByWorkTime1 := _t116;
tonToStart5(IN := start2 AND _t116, PT := _t182);
startByWorkTime2 := tonToStart5.Q;
Pump1MainDetector(CLK := pump1Main);
_en121 := Pump1MainDetector.Q;
IF _en121 THEN _t121 := FALSE; END_IF;
IF _en121 THEN pump2MainActive := _t121; END_IF;
IF _en121 THEN byCounterActive := _t121; END_IF;
IF _en121 THEN byWorkTimeActive := _t121; END_IF;
IF _en121 THEN pump3MainActive := _t121; END_IF;
Pump2MainDetector(CLK := pump2Main);
_en128 := Pump2MainDetector.Q;
IF _en128 THEN _t128 := FALSE; END_IF;
IF _en128 THEN pump1MainActive := _t128; END_IF;
IF _en128 THEN byCounterActive := _t128; END_IF;
IF _en128 THEN byWorkTimeActive := _t128; END_IF;
IF _en128 THEN pump3MainActive := _t128; END_IF;
Pump3MainDetector(CLK := pump3Main);
_en159 := Pump3MainDetector.Q;
IF _en159 THEN _t159 := FALSE; END_IF;
IF _en159 THEN pump1MainActive := _t159; END_IF;
IF _en159 THEN byCounterActive := _t159; END_IF;
IF _en159 THEN byWorkTimeActive := _t159; END_IF;
IF _en159 THEN pump2MainActive := _t159; END_IF;
ByCounterDetector(CLK := byCounter);
_en135 := ByCounterDetector.Q;
IF _en135 THEN _t135 := FALSE; END_IF;
IF _en135 THEN pump1MainActive := _t135; END_IF;
IF _en135 THEN pump2MainActive := _t135; END_IF;
IF _en135 THEN byWorkTimeActive := _t135; END_IF;
IF _en135 THEN pump3MainActive := _t135; END_IF;
ByWorkTimeDetector(CLK := byWorkTime);
_en142 := ByWorkTimeDetector.Q;
IF _en142 THEN _t142 := FALSE; END_IF;
IF _en142 THEN pump1MainActive := _t142; END_IF;
IF _en142 THEN pump2MainActive := _t142; END_IF;
IF _en142 THEN byCounterActive := _t142; END_IF;
IF _en142 THEN pump3MainActive := _t142; END_IF;
_t197 := tonToStart1.Q OR (pump2RStrig.Q1 AND start1);
_t198 := tonToStart3.Q OR (pump1RStrig.Q1 AND start1);
END_FUNCTION_BLOCK

(* POU StartLessFromThree, ST *)
FUNCTION_BLOCK StartLessFromThree
VAR_INPUT
	start1: BOOL;
	start2: BOOL;
	numberOne: UDINT;
	numberTwo: UDINT;
	numberThree: UDINT;
END_VAR
VAR_OUTPUT
	startOne: BOOL;
	startTwo: BOOL;
	startThree: BOOL;
END_VAR
VAR
	flag1: BOOL := FALSE;
	flag2: BOOL := FALSE;
	starter: UINT;
END_VAR
IF start1 = TRUE THEN

	IF flag1= FALSE THEN

		IF numberOne  <=  numberTwo AND numberOne <= numberThree THEN
			starter := 0;
			flag1 := TRUE;
		END_IF
		
		IF flag1 = FALSE AND  numberTwo  <=  numberOne AND numberTwo <= numberThree THEN
			starter := 1;
			flag1 := TRUE;
		END_IF
		
		IF flag1 = FALSE AND numberThree  <=  numberOne AND numberThree <= numberTwo THEN
			starter := 2;
			flag1 := TRUE;
		END_IF

	END_IF

	CASE starter OF
		0: startOne := TRUE;
		1: startTwo := TRUE;
		2: startThree := TRUE;
	ELSE
		startOne := FALSE;
		startTwo := FALSE;
		startThree := FALSE;
	END_CASE

		IF start2 = TRUE THEN
			IF flag2 = FALSE THEN
				CASE starter OF
					0:   IF numberTwo <= numberThree THEN
							startTwo := TRUE;
							flag2 := TRUE;
						ELSE
							startThree := TRUE;
							flag2 := TRUE;
						END_IF
					1:   IF numberOne <= numberThree THEN
							startOne := TRUE;
							flag2 := TRUE;
						ELSE
							startThree := TRUE;
							flag2 := TRUE;
						END_IF
					2:   IF numberOne <= numberTwo THEN
							startOne := TRUE;
							flag2 := TRUE;
						ELSE
							startTwo := TRUE;
							flag2 := TRUE;
						END_IF
				END_CASE
			END_IF
		ELSE
			CASE starter OF
				0:   startOne := TRUE;
					startTwo := FALSE;
					startThree := FALSE;
					flag2 := FALSE;
				1:   startTwo := TRUE;
					startOne := FALSE;
					startThree := FALSE;
					flag2 := FALSE;
				2:   startThree := TRUE;
					startOne := FALSE;
					startTwo := FALSE;
					flag2 := FALSE;
			ELSE
				startOne := FALSE;
				startTwo := FALSE;
				startThree := FALSE;
	END_CASE
		END_IF

ELSE

		startOne := FALSE;
		startTwo := FALSE;
		startThree := FALSE;
		flag1 := FALSE;

END_IF
END_FUNCTION_BLOCK

(* POU SimpleThreePump, CFC *)
FUNCTION_BLOCK SimpleThreePump
VAR_INPUT
	start1: BOOL; (*сигнал на пуск насоса 1*)
	start2: BOOL; (*сигнал на пуск насоса 2*)
	start3: BOOL; (*сигнал на пуск насоса 3*)
	alarm1: BOOL; (*авария насоса 1*)
	alarm2: BOOL; (*авария насоса 2*)
	alarm3: BOOL; (*авария насоса 3*)
END_VAR
VAR_OUTPUT
	started1: BOOL; (*сигнал на запуск насоса 1*)
	started2: BOOL; (*сигнал на запуск насоса 2*)
	started3: BOOL; (*сигнал на запуск насоса 3*)
END_VAR
VAR
	pump1changer: BOOL;
	pump2changer: BOOL;
	pump3changer: BOOL;
END_VAR
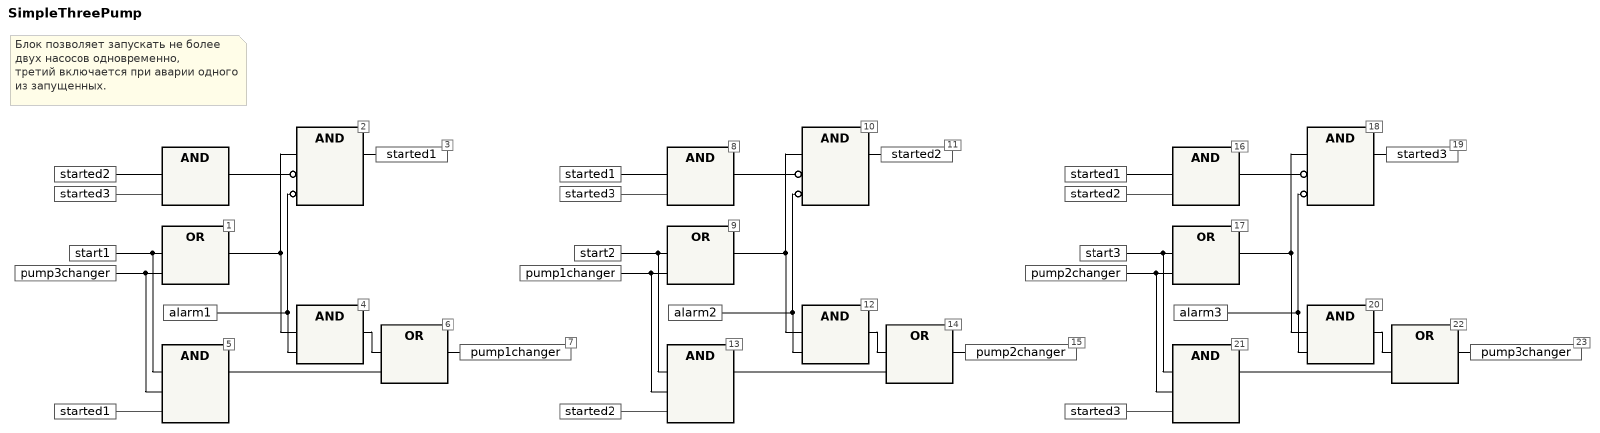
_CFC_ (* Continuous Function Chart, elements in execution order *)
#0 AND(started2, started3)
#1 OR(start1, pump3changer)
(* Блок позволяет запускать не более / двух насосов одновременно, / третий включается при аварии одного / из запущенных. *)
#2 AND(#1, NOT #0, NOT alarm1)
#3 started1 <= #2
#4 AND(#1, alarm1)
#5 AND(start1, pump3changer, started1)
#6 OR(#4, #5)
#7 pump1changer <= #6
#8 AND(started1, started3)
#9 OR(start2, pump1changer)
#10 AND(#9, NOT #8, NOT alarm2)
#11 started2 <= #10
#12 AND(#9, alarm2)
#13 AND(start2, pump1changer, started2)
#14 OR(#12, #13)
#15 pump2changer <= #14
#16 AND(started1, started2)
#17 OR(start3, pump2changer)
#18 AND(#17, NOT #16, NOT alarm3)
#19 started3 <= #18
#20 AND(#17, alarm3)
#21 AND(start3, pump2changer, started3)
#22 OR(#20, #21)
#23 pump3changer <= #22
_END_CFC_
(* the same logic as Structured Text *)
(* Блок позволяет запускать не более / двух насосов одновременно, / третий включается при аварии одного / из запущенных. *)
started1 := (start1 OR pump3changer) AND NOT (started2 AND started3) AND NOT alarm1;
pump1changer := ((start1 OR pump3changer) AND alarm1) OR (start1 AND pump3changer AND started1);
started2 := (start2 OR pump1changer) AND NOT (started1 AND started3) AND NOT alarm2;
pump2changer := ((start2 OR pump1changer) AND alarm2) OR (start2 AND pump1changer AND started2);
started3 := (start3 OR pump2changer) AND NOT (started1 AND started2) AND NOT alarm3;
pump3changer := ((start3 OR pump2changer) AND alarm3) OR (start3 AND pump2changer AND started3);
END_FUNCTION_BLOCK

(* POU FastRepeatedStartProtection, CFC *)
FUNCTION_BLOCK FastRepeatedStartProtection
VAR_INPUT
	startIN: BOOL;
	delayTime: UINT := 300;		(*время задержки, сек*)
END_VAR
VAR_OUTPUT
	startOUT: BOOL;
	SecToNextStart: UINT;		(*осталось до следующего запуска, сек*)
END_VAR
VAR
	stopDetector: F_TRIG;
	antiFreqStartTimer: TOF;
END_VAR
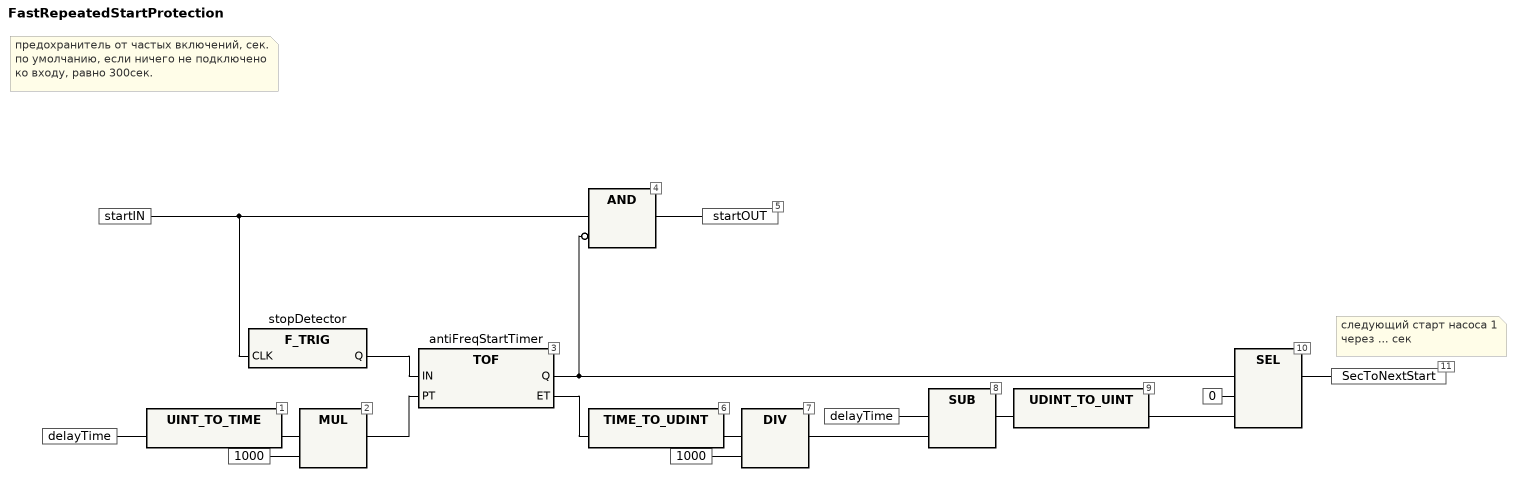
_CFC_ (* Continuous Function Chart, elements in execution order *)
(* предохранитель от частых включений, сек. / по умолчанию, если ничего не подключено / ко входу, равно 300сек. *)
(* cледующий старт насоса 1 / через ... сек *)
#0 stopDetector:F_TRIG(CLK: startIN)
#1 UINT_TO_TIME(delayTime)
#2 MUL(#1, 1000)
#3 antiFreqStartTimer:TOF(IN: #0.Q, PT: #2)
#4 AND(startIN, NOT #3.Q)
#5 startOUT <= #4
#6 TIME_TO_UDINT(#3.ET)
#7 DIV(#6, 1000)
#8 SUB(delayTime, #7)
#9 UDINT_TO_UINT(#8)
#10 SEL(#3.Q, 0, #9)
#11 SecToNextStart <= #10
_END_CFC_
(* the same logic as Structured Text *)
(* предохранитель от частых включений, сек. / по умолчанию, если ничего не подключено / ко входу, равно 300сек. *)
(* cледующий старт насоса 1 / через ... сек *)
stopDetector(CLK := startIN);
antiFreqStartTimer(IN := stopDetector.Q, PT := UINT_TO_TIME(delayTime) * 1000);
startOUT := startIN AND NOT antiFreqStartTimer.Q;
SecToNextStart := SEL(antiFreqStartTimer.Q, 0, UDINT_TO_UINT(delayTime - (TIME_TO_UDINT(antiFreqStartTimer.ET) / 1000)));
END_FUNCTION_BLOCK

(* POU PulsePerSec, CFC *)
FUNCTION_BLOCK PulsePerSec
VAR_INPUT
	start: BOOL;		(*Включает генератор импульсов.*)
END_VAR
VAR_OUTPUT
	out: BOOL;		(*Выход генератора импульсов. Начинает с FALSE.
			Каждую секунду выдает BOOL: TRUE.*)
END_VAR
VAR
	pulserRtrig: R_TRIG;		(*Детектор переднего фронта подачи импульсов.*)
	pulserRTC: RTC;		(*Таймер реального времени.*)
END_VAR
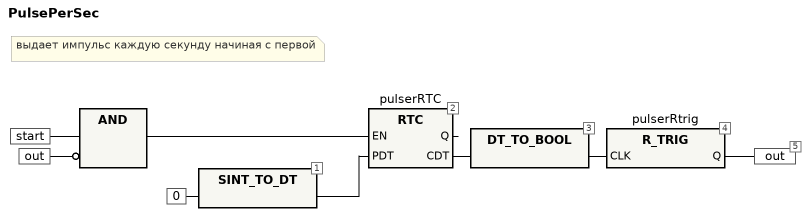
_CFC_ (* Continuous Function Chart, elements in execution order *)
(* выдает импульс каждую секунду начиная с первой *)
#0 AND(start, NOT out)
#1 SINT_TO_DT(0)
#2 pulserRTC:RTC(EN: #0, PDT: #1)
#3 DT_TO_BOOL(#2.CDT)
#4 pulserRtrig:R_TRIG(CLK: #3)
#5 out <= #4.Q
_END_CFC_
(* the same logic as Structured Text *)
(* выдает импульс каждую секунду начиная с первой *)
pulserRTC(EN := start AND NOT out, PDT := SINT_TO_DT(0));
pulserRtrig(CLK := DT_TO_BOOL(pulserRTC.CDT));
out := pulserRtrig.Q;
END_FUNCTION_BLOCK

(* POU ImpulsCounter, CFC *)
FUNCTION_BLOCK ImpulsCounter
VAR
	ImpulsDetector: R_TRIG;		(*Триггер переднего фронта входящего импульса.*)
END_VAR
VAR_INPUT
	input: BOOL;		(*Вход для импульсов, которые надо сосчитать.*)
	reset: BOOL;		(*Сброс счетчика.*)
END_VAR
VAR_OUTPUT
	countedValue: UDINT;		(*Суммарное количество импульсов.*)
END_VAR
VAR (* helpers for the ST form of the networks *)
	_t8 : UDINT;
END_VAR
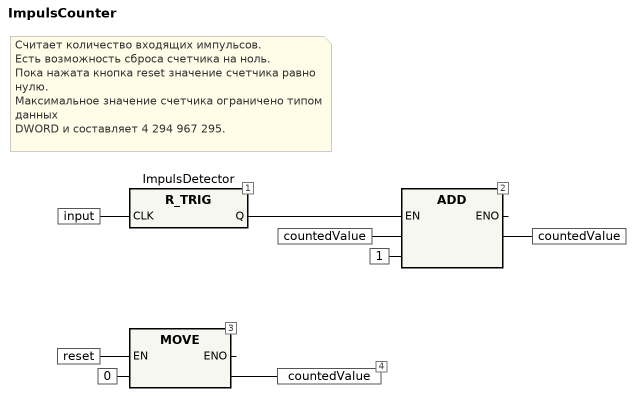
_CFC_ (* Continuous Function Chart, elements in execution order *)
(* Считает количество входящих импульсов. / Есть возможность сброса счетчика на ноль. / Пока нажата кнопка reset значение счетчика равно нулю. / Максимальное значение счетчика ограничено типом данных / DWORD и составляет 4 294 967 295. *)
#0 countedValue <= #2
#1 ImpulsDetector:R_TRIG(CLK: input)
#2 ADD(EN: #1.Q, countedValue, 1)
#3 MOVE(EN: reset, 0)
#4 countedValue <= #3
_END_CFC_
(* the same logic as Structured Text *)
(* Считает количество входящих импульсов. / Есть возможность сброса счетчика на ноль. / Пока нажата кнопка reset значение счетчика равно нулю. / Максимальное значение счетчика ограничено типом данных / DWORD и составляет 4 294 967 295. *)
countedValue := _t8;
ImpulsDetector(CLK := input);
IF ImpulsDetector.Q THEN _t8 := countedValue + 1; END_IF;
IF reset THEN countedValue := 0; END_IF;
END_FUNCTION_BLOCK

(* POU TimeSeparator, ST *)
FUNCTION_BLOCK TimeSeparator
VAR_INPUT
	 input: UDINT; (*Вход счетчика  наработки и т.п., сек.*)
END_VAR
VAR_OUTPUT
	days: UINT; (*Выход наработка, дней*)
	hours: UINT; (*Выход наработка, часов*)
	minutes: UINT; (*Выход наработка, минут*)
	seconds: UINT; (*Выход наработка, секунд*)
END_VAR
VAR
	temp: UDINT;
END_VAR
days:= UDINT_TO_INT (input / (60 * 60 * 24));
temp:= input MOD (60 * 60 * 24);
hours:= UDINT_TO_INT (temp / (60 * 60));
temp:= temp MOD (60 * 60);
minutes:= UDINT_TO_INT (temp / 60);
temp:= temp MOD 60;
seconds:= UDINT_TO_INT (temp);
END_FUNCTION_BLOCK

(* POU ChoosePumpRegime, CFC *)
FUNCTION_BLOCK ChoosePumpRegime
VAR
	pump1RStrig: RS;		(*Триггер-защелка выбора режима с главным первым насосом.*)
	pump2RStrig: RS;		(*Триггер-защелка выбора режима с главным вторым насосом.*)
	byCounterRStrig: RS;		(*Триггер-защелка выбора режима с запуском по количеству включений.*)
	byWorkTimeRStrig: RS;		(*Триггер-защелка выбора режима с запуском по наработке.*)
	Pump1MainDetector: R_TRIG;		(*Детектор переднего фронта включения режима, когда главный насос - первый.
Для сброса остальных значений.*)
	Pump2MainDetector: R_TRIG;		(*Детектор переднего фронта включения режима, когда главный насос - второй.
Для сброса остальных значений.*)
	ByCounterDetector: R_TRIG;		(*Детектор переднего фронта включения режима по количеству включений.
Для сброса остальных значений.*)
	ByWorkTimeDetector: R_TRIG;		(*Детектор переднего фронта включения режима по наработке.
Для сброса остальных значений.*)
END_VAR
VAR_INPUT
	start: BOOL;		(*Сигнал на включение насоса.
Активируется выход согласно выбранного режима.*)
	pump1Main: BOOL;		(*Режим: первый насос главный, второй - резервный.
Включать импульсом. Включать импульсом.*)
	pump2Main: BOOL;		(*Режим: второй насос главный, первый - резервный.
Включать импульсом. Включать импульсом.*)
	byCounter: BOOL;		(*Режим: запуск по количеству включений.
Включится с меньшим количеством стартов. Включать импульсом.*)
	byWorkTime: BOOL;		(*Режим: запуск по наработке.
Включится насос с меньшей наработкой. Включать импульсом.*)
END_VAR
VAR_OUTPUT
	pump1MainActive: BOOL;		(*Активный режим: первый насос главный.*)
	pump2MainActive: BOOL;		(*Активный режим: второй насос главный.*)
	byCounterActive: BOOL;		(*Активный режим: включение по количеству запусков.*)
	byWorkTimeActive: BOOL;		(*Активный режим: по наработке.*)
	startPump1: BOOL;		(*Запуск первого насоса как главного (основного).*)
	startPump2: BOOL;		(*Запуск второго насоса как главного (основного).*)
	startByCounter: BOOL;		(*Запуск насоса по количеству стартов.
			Запустится с меньшим. Если одинаково, то - первый.*)
	startByWorkTime: BOOL;		(*Запуск по наработке.
			Включится с меньшей. Если одинаково, то - первый.*)
END_VAR
VAR (* helpers for the ST form of the networks *)
	_en62 : BOOL;
	_t62 : BOOL;
	_en72 : BOOL;
	_t72 : BOOL;
	_en78 : BOOL;
	_t78 : BOOL;
	_en84 : BOOL;
	_t84 : BOOL;
END_VAR
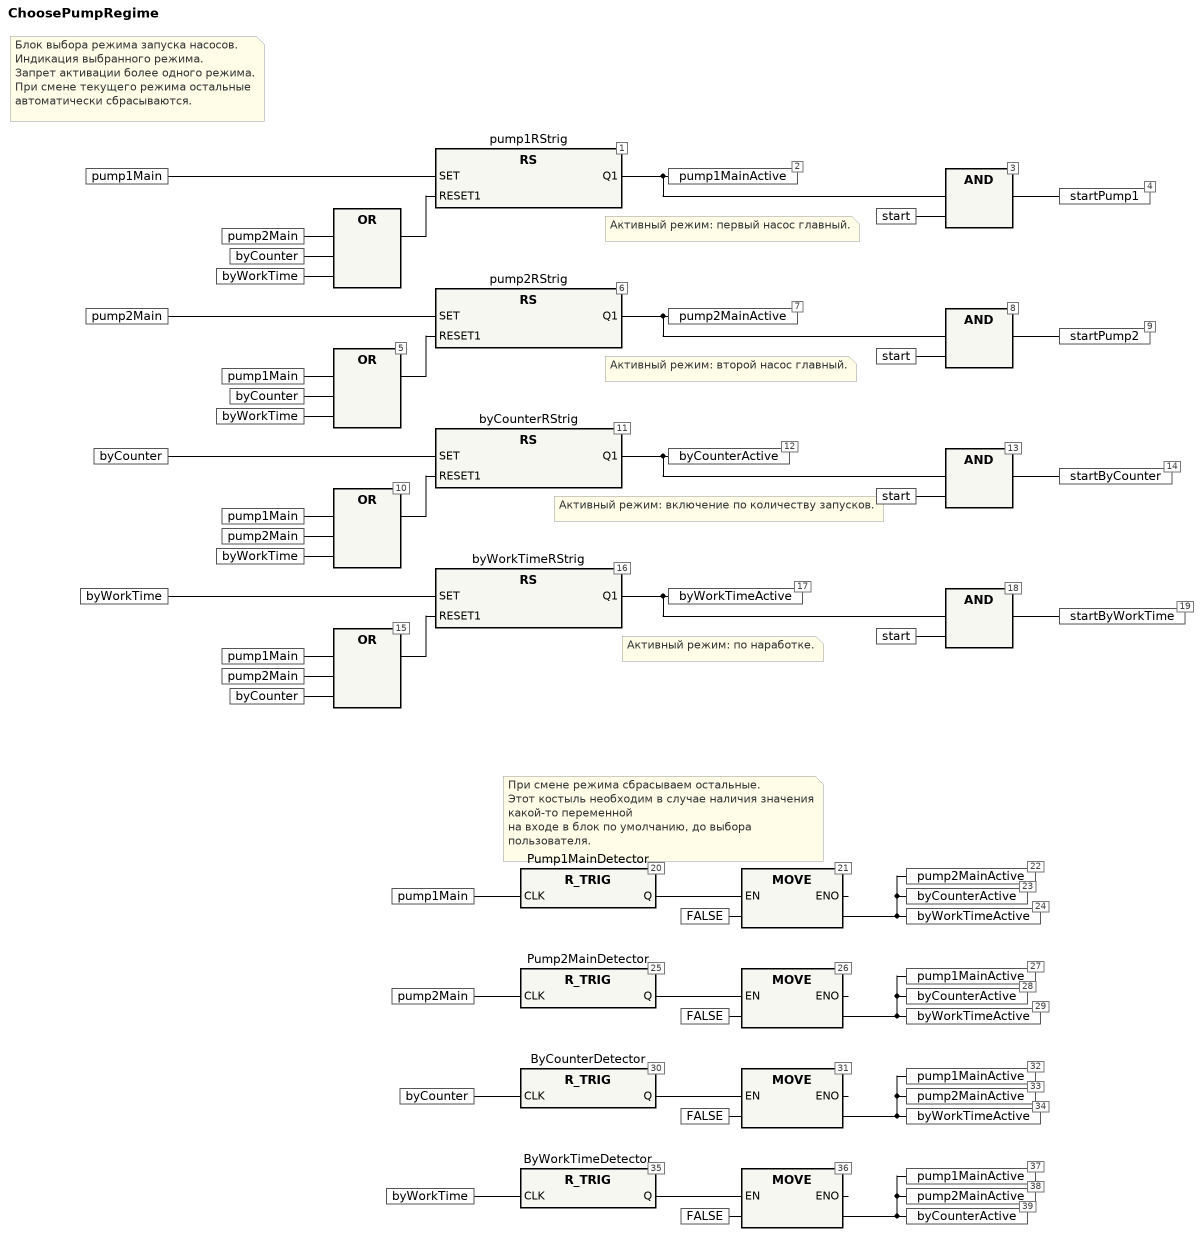
_CFC_ (* Continuous Function Chart, elements in execution order *)
(* При смене режима сбрасываем остальные. / Этот костыль необходим в случае наличия значения какой-то переменной / на входе в блок по умолчанию, до выбора пользователя. *)
(* Активный режим: второй насос главный. *)
(* Активный режим: по наработке. *)
(* Активный режим: включение по количеству запусков. *)
(* Активный режим: первый насос главный. *)
(* Блок выбора режима запуска насосов. / Индикация выбранного режима. / Запрет активации более одного режима. / При смене текущего режима остальные автоматически сбрасываются. *)
#0 OR(pump2Main, byCounter, byWorkTime)
#1 pump1RStrig:RS(SET: pump1Main, RESET1: #0)
#2 pump1MainActive <= #1.Q1
#3 AND(#1.Q1, start)
#4 startPump1 <= #3
#5 OR(pump1Main, byCounter, byWorkTime)
#6 pump2RStrig:RS(SET: pump2Main, RESET1: #5)
#7 pump2MainActive <= #6.Q1
#8 AND(#6.Q1, start)
#9 startPump2 <= #8
#10 OR(pump1Main, pump2Main, byWorkTime)
#11 byCounterRStrig:RS(SET: byCounter, RESET1: #10)
#12 byCounterActive <= #11.Q1
#13 AND(#11.Q1, start)
#14 startByCounter <= #13
#15 OR(pump1Main, pump2Main, byCounter)
#16 byWorkTimeRStrig:RS(SET: byWorkTime, RESET1: #15)
#17 byWorkTimeActive <= #16.Q1
#18 AND(#16.Q1, start)
#19 startByWorkTime <= #18
#20 Pump1MainDetector:R_TRIG(CLK: pump1Main)
#21 MOVE(EN: #20.Q, FALSE)
#22 pump2MainActive <= #21
#23 byCounterActive <= #21
#24 byWorkTimeActive <= #21
#25 Pump2MainDetector:R_TRIG(CLK: pump2Main)
#26 MOVE(EN: #25.Q, FALSE)
#27 pump1MainActive <= #26
#28 byCounterActive <= #26
#29 byWorkTimeActive <= #26
#30 ByCounterDetector:R_TRIG(CLK: byCounter)
#31 MOVE(EN: #30.Q, FALSE)
#32 pump1MainActive <= #31
#33 pump2MainActive <= #31
#34 byWorkTimeActive <= #31
#35 ByWorkTimeDetector:R_TRIG(CLK: byWorkTime)
#36 MOVE(EN: #35.Q, FALSE)
#37 pump1MainActive <= #36
#38 pump2MainActive <= #36
#39 byCounterActive <= #36
_END_CFC_
(* the same logic as Structured Text *)
(* При смене режима сбрасываем остальные. / Этот костыль необходим в случае наличия значения какой-то переменной / на входе в блок по умолчанию, до выбора пользователя. *)
(* Активный режим: второй насос главный. *)
(* Активный режим: по наработке. *)
(* Активный режим: включение по количеству запусков. *)
(* Активный режим: первый насос главный. *)
(* Блок выбора режима запуска насосов. / Индикация выбранного режима. / Запрет активации более одного режима. / При смене текущего режима остальные автоматически сбрасываются. *)
pump1RStrig(SET := pump1Main, RESET1 := pump2Main OR byCounter OR byWorkTime);
pump1MainActive := pump1RStrig.Q1;
startPump1 := pump1RStrig.Q1 AND start;
pump2RStrig(SET := pump2Main, RESET1 := pump1Main OR byCounter OR byWorkTime);
pump2MainActive := pump2RStrig.Q1;
startPump2 := pump2RStrig.Q1 AND start;
byCounterRStrig(SET := byCounter, RESET1 := pump1Main OR pump2Main OR byWorkTime);
byCounterActive := byCounterRStrig.Q1;
startByCounter := byCounterRStrig.Q1 AND start;
byWorkTimeRStrig(SET := byWorkTime, RESET1 := pump1Main OR pump2Main OR byCounter);
byWorkTimeActive := byWorkTimeRStrig.Q1;
startByWorkTime := byWorkTimeRStrig.Q1 AND start;
Pump1MainDetector(CLK := pump1Main);
_en62 := Pump1MainDetector.Q;
IF _en62 THEN _t62 := FALSE; END_IF;
IF _en62 THEN pump2MainActive := _t62; END_IF;
IF _en62 THEN byCounterActive := _t62; END_IF;
IF _en62 THEN byWorkTimeActive := _t62; END_IF;
Pump2MainDetector(CLK := pump2Main);
_en72 := Pump2MainDetector.Q;
IF _en72 THEN _t72 := FALSE; END_IF;
IF _en72 THEN pump1MainActive := _t72; END_IF;
IF _en72 THEN byCounterActive := _t72; END_IF;
IF _en72 THEN byWorkTimeActive := _t72; END_IF;
ByCounterDetector(CLK := byCounter);
_en78 := ByCounterDetector.Q;
IF _en78 THEN _t78 := FALSE; END_IF;
IF _en78 THEN pump1MainActive := _t78; END_IF;
IF _en78 THEN pump2MainActive := _t78; END_IF;
IF _en78 THEN byWorkTimeActive := _t78; END_IF;
ByWorkTimeDetector(CLK := byWorkTime);
_en84 := ByWorkTimeDetector.Q;
IF _en84 THEN _t84 := FALSE; END_IF;
IF _en84 THEN pump1MainActive := _t84; END_IF;
IF _en84 THEN pump2MainActive := _t84; END_IF;
IF _en84 THEN byCounterActive := _t84; END_IF;
END_FUNCTION_BLOCK

(* POU ControlAI, CFC *)
FUNCTION_BLOCK ControlAI
VAR_INPUT
	in: REAL;		(*Входное значение.*)
	minValue: REAL := 0;		(*Минимальное значение на выходе при 4мА на входе.
Если ко входу ничего не подключено, то 0.*)
	maxValue: REAL;		(*Максимальное значение на выходе при 20мА на входе.*)
END_VAR
VAR_OUTPUT
	out: REAL;		(*Выходное отфильтрованное значение.*)
	error: BOOL;		(*Ошибка входа.*)
END_VAR
VAR
	LIN_TRAFO: LIN_TRAFO;		(*Блок масштабирования входной величины.*)
	FilterREAL: FilterREAL;		(*Модуль фильтрации сигнала типа REAL.*)
END_VAR
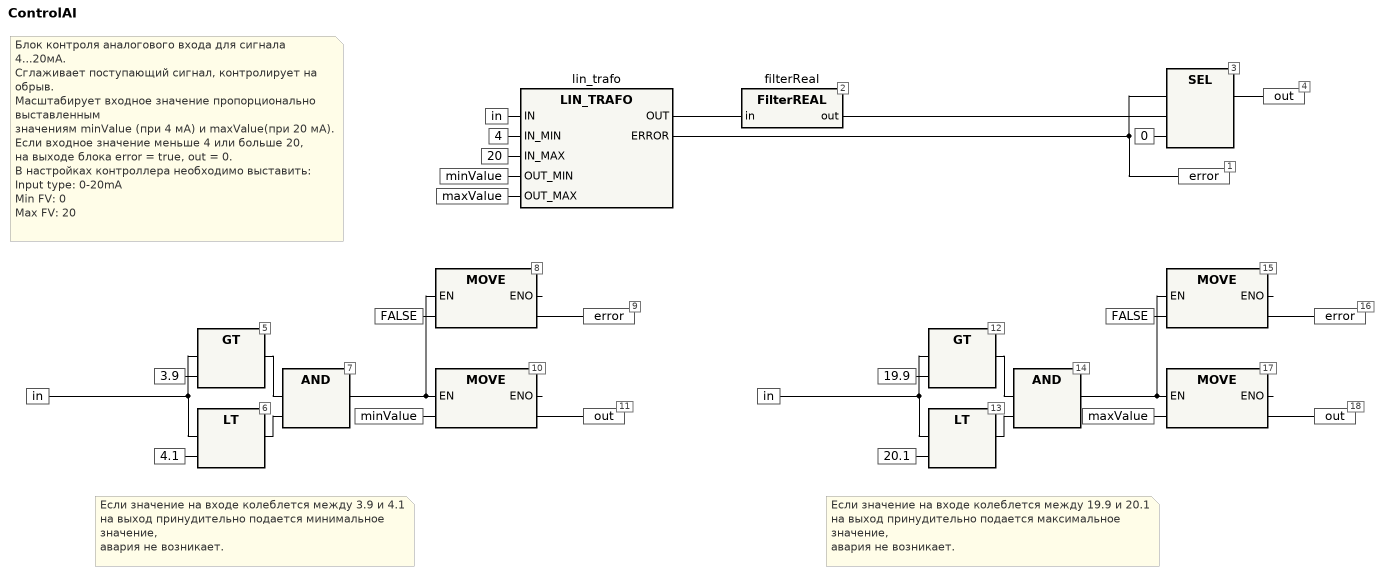
_CFC_ (* Continuous Function Chart, elements in execution order *)
(* Если значение на входе колеблется между 19.9 и 20.1 / на выход принудительно подается максимальное значение, / авария не возникает. *)
(* Если значение на входе колеблется между 3.9 и 4.1 / на выход принудительно подается минимальное значение, / авария не возникает. *)
(* Блок контроля аналогового входа для сигнала 4...20мА. / Сглаживает поступающий сигнал, контролирует на обрыв. / Масштабирует входное значение пропорционально выставленным / значениям minValue (при 4 мА) и maxValue(при 20 мА). / Если входное значение меньше 4 или больше 20, / на выходе блока error = true, out = 0. / В настройках контроллера необходимо выставить: / Input type: 0-20mA / Min FV: 0 / Max FV: 20 *)
#0 lin_trafo:LIN_TRAFO(IN: in, IN_MIN: 4, IN_MAX: 20, OUT_MIN: minValue, OUT_MAX: maxValue)
#1 error <= #0.ERROR
#2 filterReal:FilterREAL(in: #0.OUT)
#3 SEL(#0.ERROR, #2.out, 0)
#4 out <= #3
#5 GT(in, 3.9)
#6 LT(in, 4.1)
#7 AND(#5, #6)
#8 MOVE(EN: #7, FALSE)
#9 error <= #8
#10 MOVE(EN: #7, minValue)
#11 out <= #10
#12 GT(in, 19.9)
#13 LT(in, 20.1)
#14 AND(#12, #13)
#15 MOVE(EN: #14, FALSE)
#16 error <= #15
#17 MOVE(EN: #14, maxValue)
#18 out <= #17
_END_CFC_
END_FUNCTION_BLOCK

(* POU FilterREAL, ST *)
FUNCTION_BLOCK FilterREAL
VAR_INPUT
	in: REAL; (*Входное значение*)
END_VAR
VAR_OUTPUT
	out: REAL; (*Выходное значение*)
END_VAR
VAR
	k: REAL; (*Коэффициент фильтра.Чем меньше тем плавнее, чем больше, тем быстрее работает фильтр.*)
END_VAR
(*Если разница между входом и выходом больше 0,5, то коэффициент большой, фильтр - быстрый, сглаживание - минимально.*)
IF ABS(in - out) > 0.01 THEN
	k := 0.9;
ELSE
	k:=0.0001;
END_IF
out := (in - out) * k + out;
END_FUNCTION_BLOCK

(* POU CounterManager, CFC *)
FUNCTION_BLOCK CounterManager

VAR
	pump1startsCounter: ImpulsCounter;		(*Счетчик количества включений насоса 1.*)
	pump2startsCounter: ImpulsCounter;		(*Счетчик количества включений насоса 2.*)
	counterRtrig: R_TRIG;		(*Детектор переднего фронта сигнала на запуск.*)
	counterFtrig: F_TRIG;		(*Детектор спада сигнала на запуск.*)
	counterRStrigPump1: RS;		(*RSтриггер сигнала на запуск насоса 1.*)
	counterRStrigPump2: RS;		(*RSтриггер сигнала на запуск насоса 2.*)
END_VAR
VAR_INPUT
	counterStart: BOOL;		(*Сигнал на запуск насоса с наименьшей наработкой.*)
	pump1ON: BOOL;		(*Сигнал подтверждение о запуске насоса 1.*)
	pump2ON: BOOL;		(*Сигнал подтверждение о запуске насоса 2.*)
	Pump1ResetCounter: BOOL;		(*Сброс счетчика включений насоса 1.*)
	Pump2ResetCounter: BOOL;		(*Сброс счетчика включений насоса 2.*)
END_VAR
VAR_OUTPUT
	counterPump1ON: BOOL;		(*Сигнал на запуск насоса 1.*)
	counterPump2ON: BOOL;		(*Сигнал на запуск насоса 2.*)
	counterPump1: DWORD;		(*Количество включений насоса 1.*)
	counterPump2: DWORD;		(*Количество включений насоса 2.*)
END_VAR
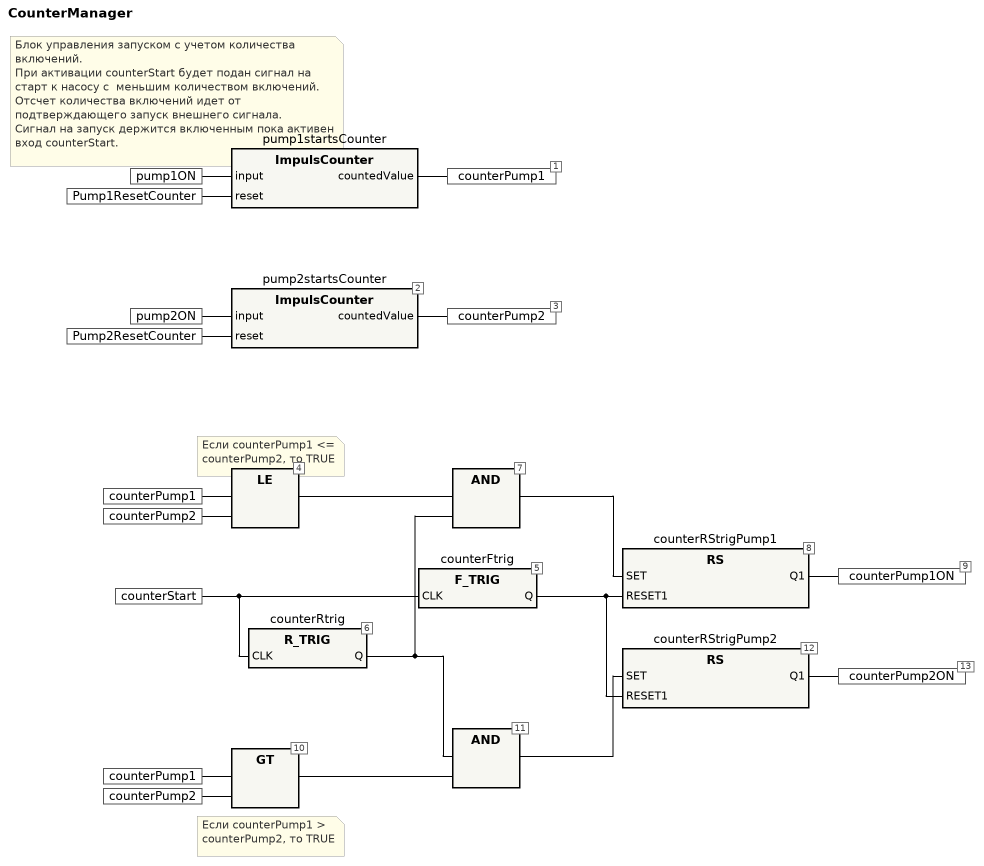
_CFC_ (* Continuous Function Chart, elements in execution order *)
(* Блок управления запуском с учетом количества включений. / При активации counterStart будет подан сигнал на старт к насосу с  меньшим количеством включений. / Отсчет количества включений идет от подтверждающего запуск внешнего сигнала. / Сигнал на запуск держится включенным пока активен вход counterStart. *)
(* Если counterPump1 <= / counterPump2, то TRUE *)
(* Если counterPump1 > / counterPump2, то TRUE *)
#0 pump1startsCounter:ImpulsCounter(input: pump1ON, reset: Pump1ResetCounter)
#1 counterPump1 <= #0.countedValue
#2 pump2startsCounter:ImpulsCounter(input: pump2ON, reset: Pump2ResetCounter)
#3 counterPump2 <= #2.countedValue
#4 LE(counterPump1, counterPump2)
#5 counterFtrig:F_TRIG(CLK: counterStart)
#6 counterRtrig:R_TRIG(CLK: counterStart)
#7 AND(#4, #6.Q)
#8 counterRStrigPump1:RS(SET: #7, RESET1: #5.Q)
#9 counterPump1ON <= #8.Q1
#10 GT(counterPump1, counterPump2)
#11 AND(#6.Q, #10)
#12 counterRStrigPump2:RS(SET: #11, RESET1: #5.Q)
#13 counterPump2ON <= #12.Q1
_END_CFC_
END_FUNCTION_BLOCK

(* POU DosingPumpProportional, CFC *)
FUNCTION_BLOCK DosingPumpProportional
VAR_INPUT
	flowValue: REAL;		(*текущее значение мгновенного расхода, кубометров в час.*)
	setMinPumpDosingValue: REAL := 0;		(*задание минимальной производительности доз.насоса.
По умолчанию, если ничего не подключено ко входу, равно нулю.*)
	setMaxPumpDosingValue: REAL;		(*задание максимальной производительности доз.насоса, в мл/мин*)
	minOutputValue: REAL := 4;		(*минимальное значение выходного сигнала.
По умолчанию, если ничего не подключено ко входу, равно 4.*)
	maxOutputValue: REAL := 20;		(*Максимально значение выходного сигнала.
По умолчанию, если ничего не подключено ко входу, равно 20.*)
	setKoeffProportionality: REAL;		(*Задание мл на кубометр (коэф.пропорциональности между расходом и дозированием)*)
	minFlowToStart: REAL := 10;		(*Минимальное значение расхода для подачи сигнала на начало дозирования.
По умолчанию, если ничего не подключено ко входу, равно 10 кубометров в час.*)
END_VAR
VAR_OUTPUT
	outputValue: REAL;		(*Выходной сигнал на дозирующий насос.*)
	dosingError: BOOL;		(*Ошибка производительности дозирования (неверно заданы значения производительности насоса, производительность доз.насоса не соответствует расходу.*)
	startDosingPump: BOOL;		(*Сигнал на запуск дозирующего насоса.*)
END_VAR
VAR
	linearTransformator: LIN_TRAFO;		(*получает на вход значение из указанного диапазона, ставит на выходе пропорциональное значение из другого диапазона.*)
END_VAR
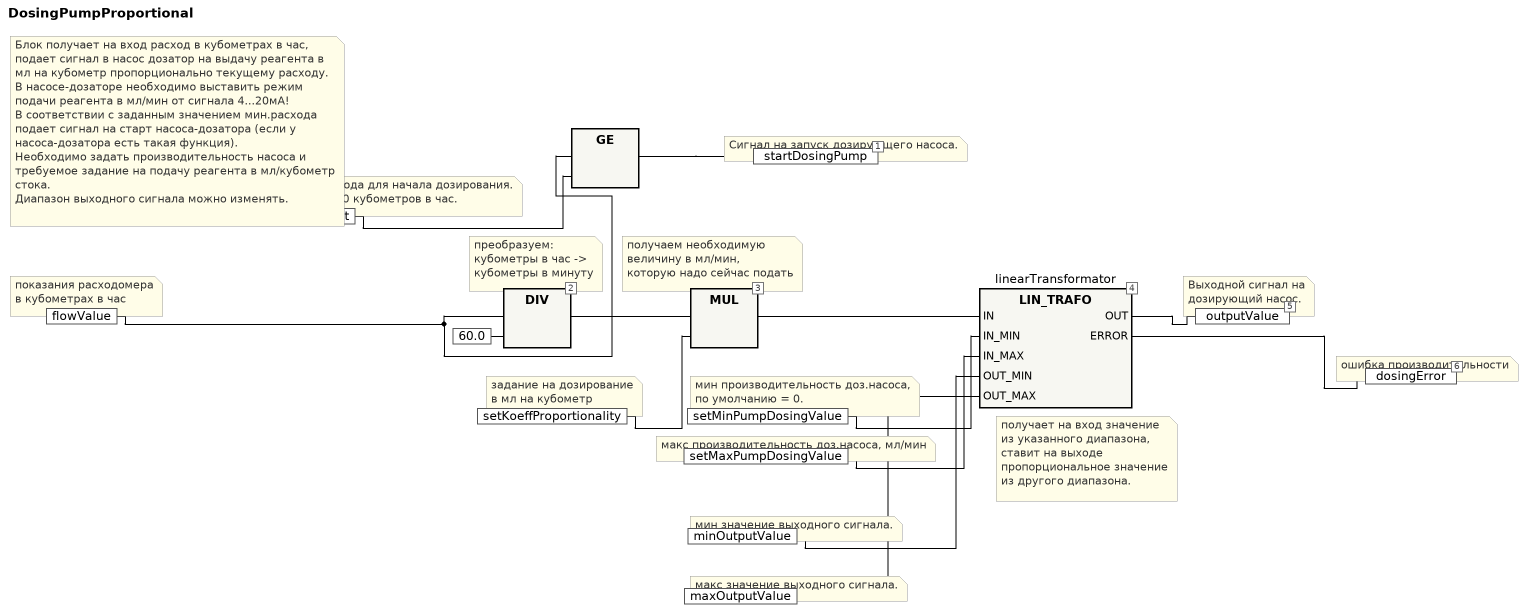
_CFC_ (* Continuous Function Chart, elements in execution order *)
(* Сигнал на запуск дозирующего насоса. *)
(* min значение расхода для начала дозирования. / По умолчанию = 10 кубометров в час. *)
(* макс производительность доз.насоса, мл/мин *)
(* мин производительность доз.насоса, / по умолчанию = 0. *)
(* получаем необходимую / величину в мл/мин, / которую надо сейчас подать *)
(* задание на дозирование / в мл на кубометр *)
(* показания расходомера / в кубометрах в час *)
(* преобразуем: / кубометры в час -> / кубометры в минуту *)
(* мин значение выходного сигнала. *)
(* макс значение выходного сигнала. *)
(* Выходной сигнал на / дозирующий насос. *)
(* ошибка производительности *)
(* получает на вход значение / из указанного диапазона, / ставит на выходе / пропорциональное значение / из другого диапазона. *)
(* Блок получает на вход расход в кубометрах в час, подает сигнал в насос дозатор на выдачу реагента в мл на кубометр пропорционально текущему расходу. / В насосе-дозаторе необходимо выставить режим подачи реагента в мл/мин от сигнала 4...20мА! / В соответствии с заданным значением мин.расхода подает сигнал на старт насоса-дозатора (если у насоса-дозатора есть такая функция). / Необходимо задать производительность насоса и требуемое задание на подачу реагента в мл/кубометр стока. / Диапазон выходного сигнала можно изменять. *)
#0 GE(flowValue, minFlowToStart)
#1 startDosingPump <= #0
#2 DIV(flowValue, 60.0)
#3 MUL(#2, setKoeffProportionality)
#4 linearTransformator:LIN_TRAFO(IN: #3, IN_MIN: setMinPumpDosingValue, IN_MAX: setMaxPumpDosingValue, OUT_MIN: minOutputValue, OUT_MAX: maxOutputValue)
#5 outputValue <= #4.OUT
#6 dosingError <= #4.ERROR
_END_CFC_
(* the same logic as Structured Text *)
(* Сигнал на запуск дозирующего насоса. *)
(* min значение расхода для начала дозирования. / По умолчанию = 10 кубометров в час. *)
(* макс производительность доз.насоса, мл/мин *)
(* мин производительность доз.насоса, / по умолчанию = 0. *)
(* получаем необходимую / величину в мл/мин, / которую надо сейчас подать *)
(* задание на дозирование / в мл на кубометр *)
(* показания расходомера / в кубометрах в час *)
(* преобразуем: / кубометры в час -> / кубометры в минуту *)
(* мин значение выходного сигнала. *)
(* макс значение выходного сигнала. *)
(* Выходной сигнал на / дозирующий насос. *)
(* ошибка производительности *)
(* получает на вход значение / из указанного диапазона, / ставит на выходе / пропорциональное значение / из другого диапазона. *)
(* Блок получает на вход расход в кубометрах в час, подает сигнал в насос дозатор на выдачу реагента в мл на кубометр пропорционально текущему расходу. / В насосе-дозаторе необходимо выставить режим подачи реагента в мл/мин от сигнала 4...20мА! / В соответствии с заданным значением мин.расхода подает сигнал на старт насоса-дозатора (если у насоса-дозатора есть такая функция). / Необходимо задать производительность насоса и требуемое задание на подачу реагента в мл/кубометр стока. / Диапазон выходного сигнала можно изменять. *)
startDosingPump := flowValue >= minFlowToStart;
linearTransformator(IN := (flowValue / 60.0) * setKoeffProportionality, IN_MIN := setMinPumpDosingValue, IN_MAX := setMaxPumpDosingValue, OUT_MIN := minOutputValue, OUT_MAX := maxOutputValue);
outputValue := linearTransformator.OUT;
dosingError := linearTransformator.ERROR;
END_FUNCTION_BLOCK

(* POU FlowVolume, CFC *)
FUNCTION_BLOCK FlowVolume
VAR_INPUT
	flowValue: REAL;		(*Вход от расходомера, мгновенный расход в кубометрах в час.*)
	setVolume: REAL;		(*Контрольный объем. Сравнивается с накопленным по показаниям расходомера,
Если превышает, счетчик сбрасывается, на выход out подается импульс.
Если на входе ноль, то условие не работает, блок просто считает сумму стоков.*)
	reset: BOOL;		(*Ручной сброс счетчика.*)
END_VAR
VAR_OUTPUT
	totalAmount: REAL;		(*Сумма накопленных стоков.*)
	out: BOOL;		(*Импульс - сигнал что сумма стоков равна или больше
заданному в setVolume значению.*)
END_VAR
VAR
	pulsPerSec: PulsePerSec;		(*Генератор импульс в секунду.*)
END_VAR
VAR (* helpers for the ST form of the networks *)
	_t22 : BOOL;
END_VAR
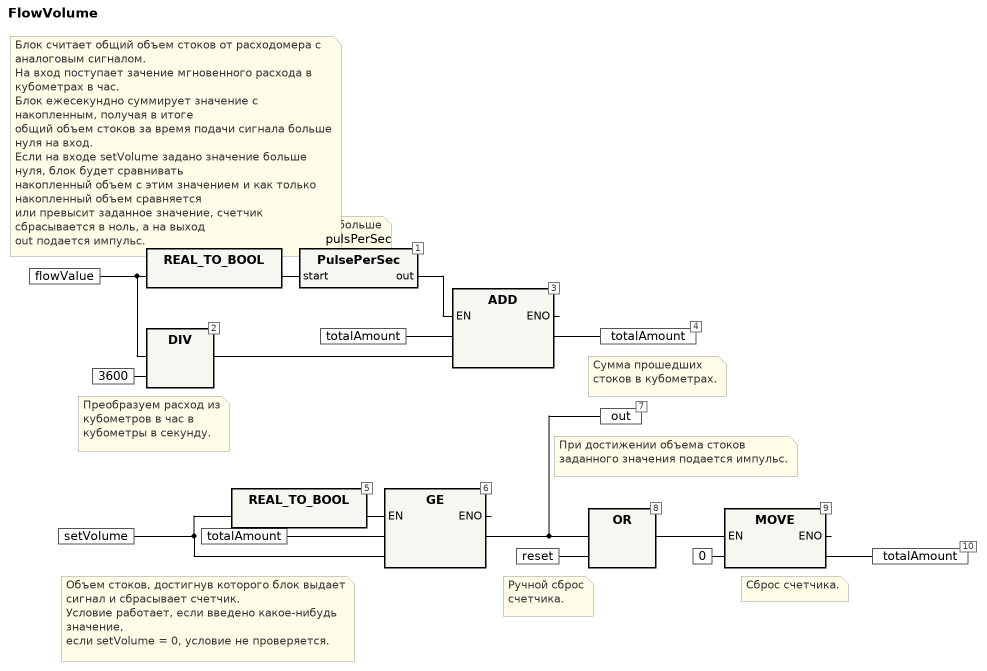
_CFC_ (* Continuous Function Chart, elements in execution order *)
(* Ручной сброс / счетчика. *)
(* При достижении объема стоков / заданного значения подается импульс. *)
(* Сумма прошедших / стоков в кубометрах. *)
(* Объем стоков, достигнув которого блок выдает / сигнал и сбрасывает счетчик. / Условие работает, если введено какое-нибудь значение, / если setVolume = 0, условие не проверяется. *)
(* Преобразуем расход из / кубометров в час в / кубометры в секунду. *)
(* Начинаем считать стоки при наличии расхода больше нуля. *)
(* Сброс счетчика. *)
(* Блок считает общий объем стоков от расходомера с аналоговым сигналом. / На вход поступает зачение мгновенного расхода в кубометрах в час. / Блок ежесекундно суммирует значение с накопленным, получая в итоге / общий объем стоков за время подачи сигнала больше нуля на вход. / Если на входе setVolume задано значение больше нуля, блок будет сравнивать / накопленный объем с этим значением и как только накопленный объем сравняется / или превысит заданное значение, счетчик сбрасывается в ноль, а на выход / out подается импульс. *)
#0 REAL_TO_BOOL(flowValue)
#1 pulsPerSec:PulsePerSec(start: #0)
#2 DIV(flowValue, 3600)
#3 ADD(EN: #1.out, totalAmount, #2)
#4 totalAmount <= #3
#5 REAL_TO_BOOL(setVolume)
#6 GE(EN: #5, totalAmount, setVolume)
#7 out <= #6
#8 OR(#6, reset)
#9 MOVE(EN: #8, 0)
#10 totalAmount <= #9
_END_CFC_
(* the same logic as Structured Text *)
(* Ручной сброс / счетчика. *)
(* При достижении объема стоков / заданного значения подается импульс. *)
(* Сумма прошедших / стоков в кубометрах. *)
(* Объем стоков, достигнув которого блок выдает / сигнал и сбрасывает счетчик. / Условие работает, если введено какое-нибудь значение, / если setVolume = 0, условие не проверяется. *)
(* Преобразуем расход из / кубометров в час в / кубометры в секунду. *)
(* Начинаем считать стоки при наличии расхода больше нуля. *)
(* Сброс счетчика. *)
(* Блок считает общий объем стоков от расходомера с аналоговым сигналом. / На вход поступает зачение мгновенного расхода в кубометрах в час. / Блок ежесекундно суммирует значение с накопленным, получая в итоге / общий объем стоков за время подачи сигнала больше нуля на вход. / Если на входе setVolume задано значение больше нуля, блок будет сравнивать / накопленный объем с этим значением и как только накопленный объем сравняется / или превысит заданное значение, счетчик сбрасывается в ноль, а на выход / out подается импульс. *)
pulsPerSec(start := REAL_TO_BOOL(flowValue));
IF pulsPerSec.out THEN totalAmount := totalAmount + (flowValue / 3600); END_IF;
IF REAL_TO_BOOL(setVolume) THEN _t22 := totalAmount >= setVolume; END_IF;
out := _t22;
IF _t22 OR reset THEN totalAmount := 0; END_IF;
END_FUNCTION_BLOCK

(* POU IfBOOL, ST *)
FUNCTION_BLOCK IfBOOL
VAR_INPUT
	key: BOOL; (*Ключ. Если TRUE, то сигнал на входе будет передан на выход keyTRUE, иначе на keyFALSE.*)
	input: BOOL; (*Вход*)
END_VAR
VAR_OUTPUT
	keyFALSE: BOOL; (*Выход  получит значение от входа, если key = FALSE.*)
	keyTRUE: BOOL; (*Выход  получит значение от входа, если key = TRUE.*)
END_VAR
VAR
END_VAR
IF key = TRUE THEN
	keyTRUE := input;
	keyFALSE := FALSE;
ELSE keyTRUE := FALSE;
		keyFALSE := input;
END_IF
END_FUNCTION_BLOCK

(* POU ImpulsFlowCounter, CFC *)
FUNCTION_BLOCK ImpulsFlowCounter
VAR_INPUT
	impulsInput: BOOL;		(*Входящие импульсы от расходомера.
Каждый импульс будет прибавлять в итоговую сумму величину веса импульса.*)
	impulsValue: REAL;		(*Вес импульса расходомера.*)
	resetCounter: BOOL;		(*Сброс счетчика.*)
	correctionValue: REAL;		(*Число, которое будет прибавлено или вычтено из накопленной суммы.*)
	addCorrection: BOOL;		(*Прибавить коррекцию к накопленной сумме.*)
	deleteCorrection: BOOL;		(*Вычесть коррекцию из накопленной суммы.
Если получится отрицательное число, сумма скинется в ноль.*)
END_VAR
VAR_OUTPUT
	totalAmountREAL: REAL;		(*Накопленная сумма в десятичном виде.
От 10 млн может выводиться в экспоненциальной форме.*)
	totalAmountDWORD: DWORD;		(*Накопленная сумма в целочисленном виде.
Округление десятичных по правилам арифметики.*)
END_VAR
VAR
	inputImpulsRtrig: R_TRIG;		(*Детектор переднего фронта входящих импульсов.*)
	resetRtrig: R_TRIG;		(*Детектор переднего фронта сигнала на сброс счетчика.*)
	addCorrRtrig: R_TRIG;		(*Детектор переднего фронта сигнала на прибавление коррекции.*)
	deleteCorrRtrig: R_TRIG;		(*Детектор переднего фронта сигнала на вычитание коррекции.*)
END_VAR
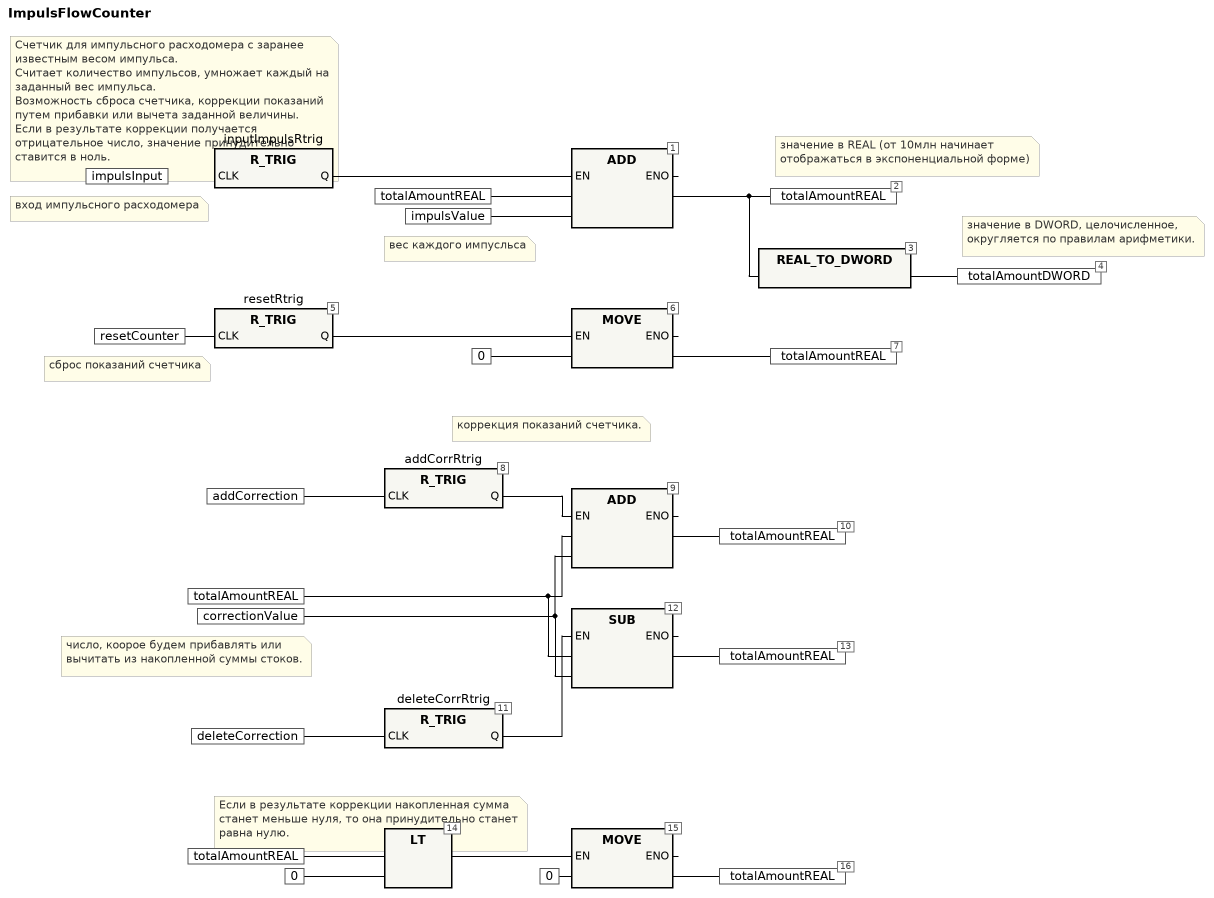
_CFC_ (* Continuous Function Chart, elements in execution order *)
(* вход импульсного расходомера *)
(* сброс показаний счетчика *)
(* значение в REAL (от 10млн начинает / отображаться в экспоненциальной форме) *)
(* значение в DWORD, целочисленное, / округляется по правилам арифметики. *)
(* Если в результате коррекции накопленная сумма станет меньше нуля, то она принудительно станет равна нулю. *)
(* коррекция показаний счетчика. *)
(* число, коорое будем прибавлять или / вычитать из накопленной суммы стоков. *)
(* вес каждого импусльса *)
(* Счетчик для импульсного расходомера с заранее известным весом импульса. / Считает количество импульсов, умножает каждый на заданный вес импульса. / Возможность сброса счетчика, коррекции показаний путем прибавки или вычета заданной величины. / Если в результате коррекции получается отрицательное число, значение принудительно ставится в ноль. *)
#0 inputImpulsRtrig:R_TRIG(CLK: impulsInput)
#1 ADD(EN: #0.Q, totalAmountREAL, impulsValue)
#2 totalAmountREAL <= #1
#3 REAL_TO_DWORD(#1)
#4 totalAmountDWORD <= #3
#5 resetRtrig:R_TRIG(CLK: resetCounter)
#6 MOVE(EN: #5.Q, 0)
#7 totalAmountREAL <= #6
#8 addCorrRtrig:R_TRIG(CLK: addCorrection)
#9 ADD(EN: #8.Q, totalAmountREAL, correctionValue)
#10 totalAmountREAL <= #9
#11 deleteCorrRtrig:R_TRIG(CLK: deleteCorrection)
#12 SUB(EN: #11.Q, totalAmountREAL, correctionValue)
#13 totalAmountREAL <= #12
#14 LT(totalAmountREAL, 0)
#15 MOVE(EN: #14, 0)
#16 totalAmountREAL <= #15
_END_CFC_
END_FUNCTION_BLOCK

